    /// <summary>PDT-02</summary>
	{attribute 'OPC.UA.DA' := '1'}  				                
	sorbent_diff_pres_low												: REAL;
    /// <summary>PDT-02</summary>
	{attribute 'OPC.UA.DA' := '1'}  				                
	sorbent_diff_pres_high												: REAL;
    /// <summary>PDT-02</summary>
	{attribute 'OPC.UA.DA' := '1'}  				                
	sorbent_diff_pres_min												: REAL;
    /// <summary>PDT-02</summary>
	{attribute 'OPC.UA.DA' := '1'}  				                
	sorbent_diff_pres_offset											: REAL;

    /// <summary>PDT-03</summary>
	{attribute 'OPC.UA.DA' := '1'}  				                
	fan_diff_pres_low													: REAL;
    /// <summary>PDT-03</summary>
	{attribute 'OPC.UA.DA' := '1'}  				                
	fan_diff_pres_high													: REAL;
    /// <summary>PDT-03</summary>
	{attribute 'OPC.UA.DA' := '1'}  				                
	fan_diff_pres_min													: REAL;
    /// <summary>PDT-03</summary>
	{attribute 'OPC.UA.DA' := '1'}  				                
	fan_diff_pres_offset												: REAL;

    /// <summary>PT-01</summary>
	{attribute 'OPC.UA.DA' := '1'}  				                
	reactor_pres_low													: REAL;
    /// <summary>PT-01</summary>
	{attribute 'OPC.UA.DA' := '1'}  				                
	reactor_pres_high													: REAL;
    /// <summary>PT-01</summary>
	{attribute 'OPC.UA.DA' := '1'}  				                
	reactor_pres_min													: REAL;
    /// <summary>PT-01</summary>
	{attribute 'OPC.UA.DA' := '1'}  				                
	reactor_pres_offset													: REAL;

    /// <summary>TT-05</summary>
	{attribute 'OPC.UA.DA' := '1'}  				                
	reactor_wall_temp_offset											: REAL;

    /// <summary>TT-06</summary>
	{attribute 'OPC.UA.DA' := '1'}  				                
	outlet_line_temp_offset												: REAL;

	
    /// <summary>01-TT-01</summary>
	{attribute 'OPC.UA.DA' := '1'}  				                
	cart01_front_temp_offset											: REAL;
    /// <summary>10-TT-03</summary>
	{attribute 'OPC.UA.DA' := '1'}  				                
	cart01_back_temp_offset												: REAL;
    /// <summary>02-TT-01</summary>
	{attribute 'OPC.UA.DA' := '1'}  				                
	cart02_front_temp_offset											: REAL;
    /// <summary>02-TT-03</summary>
	{attribute 'OPC.UA.DA' := '1'}  				                
	cart02_back_temp_offset												: REAL;
    /// <summary>03-TT-01</summary>
	{attribute 'OPC.UA.DA' := '1'}  				                
	cart03_front_temp_offset											: REAL;
    /// <summary>03-TT-03</summary>
	{attribute 'OPC.UA.DA' := '1'}  				                
	cart03_back_temp_offset												: REAL;
    /// <summary>04-TT-01</summary>
	{attribute 'OPC.UA.DA' := '1'}  				                
	cart04_front_temp_offset											: REAL;
    /// <summary>04-TT-03</summary>
	{attribute 'OPC.UA.DA' := '1'}  				                
	cart04_back_temp_offset												: REAL;
    /// <summary>05-TT-01</summary>
	{attribute 'OPC.UA.DA' := '1'}  				                
	cart05_front_temp_offset											: REAL;
    /// <summary>05-TT-03</summary>
	{attribute 'OPC.UA.DA' := '1'}  				                
	cart05_back_temp_offset												: REAL;
    /// <summary>06-TT-01</summary>
	{attribute 'OPC.UA.DA' := '1'}  				                
	cart06_front_temp_offset											: REAL;
    /// <summary>06-TT-03</summary>
	{attribute 'OPC.UA.DA' := '1'}  				                
	cart06_back_temp_offset												: REAL;
    /// <summary>07-TT-01</summary>
	{attribute 'OPC.UA.DA' := '1'}  				                
	cart07_front_temp_offset											: REAL;
    /// <summary>07-TT-03</summary>
	{attribute 'OPC.UA.DA' := '1'}  				                
	cart07_back_temp_offset												: REAL;
    /// <summary>08-TT-01</summary>
	{attribute 'OPC.UA.DA' := '1'}  				                
	cart08_front_temp_offset											: REAL;
    /// <summary>08-TT-03</summary>
	{attribute 'OPC.UA.DA' := '1'}  				                
	cart08_back_temp_offset												: REAL;
    /// <summary>09-TT-01</summary>
	{attribute 'OPC.UA.DA' := '1'}  				                
	cart09_front_temp_offset											: REAL;
    /// <summary>09-TT-03</summary>
	{attribute 'OPC.UA.DA' := '1'}  				                
	cart09_back_temp_offset												: REAL;
    /// <summary>10-TT-01</summary>
	{attribute 'OPC.UA.DA' := '1'}  				                
	cart10_front_temp_offset											: REAL;
    /// <summary>10-TT-03</summary>
	{attribute 'OPC.UA.DA' := '1'}  				                
	cart10_back_temp_offset												: REAL;
    /// <summary>11-TT-01</summary>
	{attribute 'OPC.UA.DA' := '1'}  				                
	cart11_front_temp_offset											: REAL;
    /// <summary>11-TT-03</summary>
	{attribute 'OPC.UA.DA' := '1'}  				                
	cart11_back_temp_offset												: REAL;
    /// <summary>12-TT-01</summary>
	{attribute 'OPC.UA.DA' := '1'}  				                
	cart12_front_temp_offset											: REAL;
    /// <summary>12-TT-03</summary>
	{attribute 'OPC.UA.DA' := '1'}  				                
	cart12_back_temp_offset												: REAL;
	
END_VAR

// ---- GVLs/P0_Global_Variables.TcGVL
// Phase 0 - Global_Variables
// Rev 1.0 - May 11, 2024

VAR_GLOBAL

	sita_bits															: ARRAY[1..10] OF DINT;
	
	

	gbRS01TestError														: BOOL;
	gbRS02TestError														: BOOL;
	gbRS03TestError														: BOOL;
	
	gbDrainageOn														: BOOL;
	gbSafeShutdownRunning												: BOOL;

	giEvacuationErrorRS													: INT		:= 0;
	giDesorptionErrorRS													: INT		:= 0;
	giSafeShutdown1RS													: INT		:= 0;
	giSafeShutdown23RS													: INT		:= 0;
	
	gsCycleMode															: STRING;
	gsCycleStage														: STRING;
	gsM01RS01CycleStage													: STRING;
	gsM01RS02CycleStage													: STRING;
	gsM01RS03CycleStage													: STRING;
	
// These values allow points in error to be bypassed for testing purposes
	_BoilerOutletPresOff												: BOOL		:= TRUE;// FALSE;
	_BoilerOutletTempOff                        						: BOOL		:= FALSE;
	_CondensateCollectionTankFlowOff									: BOOL		:= FALSE;
	_CondensateCollectionTankLevelOff									: BOOL		:= FALSE;
	_CondensateCollectionTankO2Off										: BOOL		:= FALSE;
	_CondensateCollectionTankOutletLineTempOff  						: BOOL		:= FALSE;
	_CondensateCollectionTankPhOff										: BOOL		:= FALSE;
	_CondensateCollectionTankTempOff            						: BOOL		:= FALSE;
	_CondensateCollectionTankTurbidityOff								: BOOL		:= FALSE;
	_DeadAirFlowOff														: BOOL		:= FALSE;
	_DeadAirLineCo2Off													: BOOL		:= FALSE;
	_DeadAirLinePresOff													: BOOL		:= FALSE;
	_InstrumentAirCompPresOff                   						: BOOL		:= FALSE;
	_InstrumentAirCompTempOff                   						: BOOL		:= TRUE;
	_PostCondenserLinePresOff											: BOOL		:= FALSE;
	_PostCondenserLineTempOff                   						: BOOL		:= FALSE;
	_PreCondenserLinePresOff											: BOOL		:= FALSE;
	_PreCondenserLineTempOff                    						: BOOL		:= FALSE;
	_ProductCondensateDrumLevelOff										: BOOL		:= FALSE;
	_ProductCondenserPumpOutlerLiquidFlowOff							: BOOL		:= FALSE;
	_ProductCondenserPumpOutletTempOff          						: BOOL		:= FALSE;
	_ProductOutletCo2Off												: BOOL		:= FALSE;
	_ProductOutletH2oOff												: BOOL		:= FALSE;
	_ProductCo2SampleH2oOff												: BOOL		:= FALSE;
	_ProductOutletTemperatureOff										: BOOL		:= FALSE;
	_ProductOutletO2Off													: BOOL		:= FALSE;
	_ProductOutletPresOff												: BOOL		:= FALSE;
	_ProductOutletTempOff                       						: BOOL		:= FALSE;
	_ProductOutMassFlowOff												: BOOL		:= FALSE;
	_ProductOutVolumetricFlowOff										: BOOL		:= FALSE;
	_ProductVacuumPresOff												: BOOL		:= FALSE;
	_PurgeProductLinePresOff											: BOOL		:= FALSE;
	_PurgeProductLineTempOff											: BOOL		:= FALSE;
	_SteamHeadFlowOff													: BOOL		:= FALSE;
	_WaterToBoilerFlowOff												: BOOL		:= FALSE;
	_WeatherHumidityOff													: BOOL		:= FALSE;
	_WeatherNoiseLevelOff												: BOOL		:= FALSE;
	_WeatherPressureOff													: BOOL		:= FALSE;
	_WeatherTempOff														: BOOL		:= FALSE;
	_WeatherWindDirectionOff											: BOOL		:= FALSE;
	_WeatherWindSpeedOff												: BOOL		:= FALSE;

	_CondensateFlowOff													: BOOL		:= FALSE;
 	_SteamManifoldLinePresOff											: BOOL		:= FALSE;
	_SteamTempNearRS01Off												: BOOL		:= FALSE;           						
	_SteamTempNearRS03Off												: BOOL		:= FALSE;           						
	_CondensateTempOff													: BOOL		:= FALSE;           						
	
END_VAR

// ---- GVLs/m01.TcGVL
// Phase 0 - m01
// Rev 1.0 - April 25, 2024

{attribute 'qualified_only'}
VAR_GLOBAL

	{attribute 'OPC.UA.DA' := '1'}  				                
	{attribute 'OPC.UA.DA.Access' := '1'}  				                
	plc_version															: STRING;

	{attribute 'OPC.UA.DA' := '1'}  				                
	ts_Cycle_Mode														: STRING;		// Starts process based on each character in integer format
	{attribute 'OPC.UA.DA' := '1'}  				                
	tb_HMI_Active														: BOOL;			// An HMI program is running and communicating
	{attribute 'OPC.UA.DA' := '1'}  				                
	tb_Acknowledge_Alarm												: BOOL;			// Clears current alarm
	{attribute 'OPC.UA.DA' := '1'}  				                
	tb_Clear_Alarm_All													: BOOL;			// Clears current alarm
	{attribute 'OPC.UA.DA' := '1'}  				                
	tb_Cancel_Cycle														: BOOL;			// Complete current cycle then stop
	{attribute 'OPC.UA.DA' := '1'}  				                
	tb_Stop_Process														: BOOL;			// Stop current process immediately
	{attribute 'OPC.UA.DA' := '1'}  				                
	tb_Reset_Process													: BOOL;
	
	{attribute 'OPC.UA.DA' := '1'}  				                
	{attribute 'OPC.UA.DA.Access' := '1'}  				                
	tb_Alarm_Active														: BOOL;			// An alarm is active
	{attribute 'OPC.UA.DA' := '1'}  				                
	{attribute 'OPC.UA.DA.Access' := '1'}  				                
	ts_Alarm															: STRING;		// Active alarm string
	{attribute 'OPC.UA.DA' := '1'}  				                
	{attribute 'OPC.UA.DA.Access' := '1'}  				                
	ts_User_Message														: STRING;		// Message corresponding to active alarm
	{attribute 'OPC.UA.DA' := '1'}  				                
	{attribute 'OPC.UA.DA.Access' := '1'}  				                
	ti_Alarm_Severity													: INT;			// Alarm level (not implemented)	
	{attribute 'OPC.UA.DA' := '1'}  
	processAlarms														: ARRAY[0.._ALARM_COUNT] OF STRING;
	{attribute 'OPC.UA.DA' := '1'}  
	processAlarmsMessage												: ARRAY[0.._ALARM_COUNT] OF STRING;
					
	{attribute 'OPC.UA.DA' := '1'}  				                
	{attribute 'OPC.UA.DA.Access' := '1'}  				                
	tb_Auto_Mode_On														: BOOL;			// Machine is currently in auto mode
	
	
	
	{attribute 'OPC.UA.DA' := '1'} 	
	dispatch_active_queue_steam_pump 									: ARRAY[1..rs_count] OF UINT;
	{attribute 'OPC.UA.DA' := '1'} 	
	dispatch_passive_queue_steam_pump 									: ARRAY[1..rs_count] OF UINT;
		{attribute 'OPC.UA.DA' := '1'} 	
	dispatch_active_queue_dead_pump 									: ARRAY[1..rs_count] OF UINT; 
	{attribute 'OPC.UA.DA' := '1'} 	
	dispatch_passive_queue_dead_pump 									: ARRAY[1..rs_count] OF UINT; 

	
    /// <summary>FT-02</summary>
	{attribute 'OPC.UA.DA' := '1'}  				                
	{attribute 'OPC.UA.DA.Access' := '1'}  				                
	condensate_flow														: REAL;
    /// <summary>FT-02</summary>
	{attribute 'OPC.UA.DA' := '1'}  				                
	{attribute 'OPC.UA.DA.Access' := '1'}  				                
	condensate_flow_error										AT %I*	: BOOL;
    /// <summary>condensate flow</summary>
	FT_02														AT %I*	: INT;

    /// <summary>PT-02</summary>
	{attribute 'OPC.UA.DA' := '1'}  				                
	{attribute 'OPC.UA.DA.Access' := '1'}  				                
	steam_manifold_line_pres											: REAL;
    /// <summary>PT-02</summary>
	{attribute 'OPC.UA.DA' := '1'}  				                
	{attribute 'OPC.UA.DA.Access' := '1'}  				                
	steam_manifold_line_pres_error								AT %I*	: BOOL;
    /// <summary>steam manifold line pres</summary>
	PT_02														AT %I*	: INT;

    /// <summary>LS-03</summary>
	{attribute 'OPC.UA.DA' := '1'}  				                
	{attribute 'OPC.UA.DA.Access' := '1'}  				                
	condensate_from_cooling_and_purge_lines_lsl					AT %I*	: BOOL;
	
    /// <summary>LS-04</summary>
	{attribute 'OPC.UA.DA' := '1'}  				                
	{attribute 'OPC.UA.DA.Access' := '1'}  				                
	condensate_from_cooling_and_purge_lines_lsh					AT %I*	: BOOL;

    /// <summary>P-02</summary>
	{attribute 'OPC.UA.DA' := '1'}  				                
	condensate_from_cooling_and_purge_lines_pump						: BOOL;
    /// <summary>P-02</summary>
	{attribute 'OPC.UA.DA' := '1'}  				                
	{attribute 'OPC.UA.DA.Access' := '1'}  				                
	condensate_from_cooling_and_purge_lines_pump_cmd_status				: BOOL;
    /// <summary>condensate from cooling and purge lines pump</summary>
	P_02														AT %Q*	: BOOL;

    /// <summary>TT-10</summary>
	{attribute 'OPC.UA.DA' := '1'}  				                
	{attribute 'OPC.UA.DA.Access' := '1'}  				                
	steam_temp_near_rs1													: REAL;
    /// <summary>TT-10</summary>
	{attribute 'OPC.UA.DA' := '1'}  				                
	{attribute 'OPC.UA.DA.Access' := '1'}  				                
	steam_temp_near_rs1_error									AT %I*	: BOOL;
    /// <summary>steam temp near rs1 error</summary>
	TT_10														AT %I*	: INT;

    /// <summary>TT-11</summary>
	{attribute 'OPC.UA.DA' := '1'}  				                
	{attribute 'OPC.UA.DA.Access' := '1'}  				                
	steam_temp_near_rs3													: REAL;
    /// <summary>TT-11</summary>
	{attribute 'OPC.UA.DA' := '1'}  				                
	{attribute 'OPC.UA.DA.Access' := '1'}  				                
	steam_temp_near_rs3_error									AT %I*	: BOOL;
    /// <summary>steam temp near rs3 error</summary>
	TT_11														AT %I*	: INT;

    /// <summary>TT-12</summary>
	{attribute 'OPC.UA.DA' := '1'}  				                
	{attribute 'OPC.UA.DA.Access' := '1'}  				                
	condensate_temp														: REAL;
    /// <summary>TT-12</summary>
	{attribute 'OPC.UA.DA' := '1'}  				                
	{attribute 'OPC.UA.DA.Access' := '1'}  				                
	condensate_temp_error										AT %I*	: BOOL;
    /// <summary>condensate temp</summary>
	TT_12														AT %I*	: INT;

	{attribute 'OPC.UA.DA' := '1'}  				                
	l1_current															: REAL;
	{attribute 'OPC.UA.DA' := '1'}  				                
	l1_current_error											AT %I*	: BOOL;
	IT_01														AT %I*	: INT;
	{attribute 'OPC.UA.DA' := '1'}  				                
	l2_current															: REAL;
	{attribute 'OPC.UA.DA' := '1'}  				                
	l2_current_error											AT %I*	: BOOL;
	IT_02														AT %I*	: INT;
	{attribute 'OPC.UA.DA' := '1'}  				                
	l3_current															: REAL;
	{attribute 'OPC.UA.DA' := '1'}  				                
	l3_current_error											AT %I*	: BOOL;
	IT_03														AT %I*	: INT;
	
	{attribute 'OPC.UA.DA' := '1'}  				                
	l1_voltage															: REAL;
	{attribute 'OPC.UA.DA' := '1'}  				                
	l1_volatge_error											AT %I*	: BOOL;
	VT_01														AT %I*	: INT;
	{attribute 'OPC.UA.DA' := '1'}  				                
	l2_voltage															: REAL;
	{attribute 'OPC.UA.DA' := '1'}  				                
	l2_volatge_error											AT %I*	: BOOL;
	VT_02														AT %I*	: INT;
	{attribute 'OPC.UA.DA' := '1'}  				                
	l3_voltage															: REAL;
	{attribute 'OPC.UA.DA' := '1'}  				                
	l3_volatge_error											AT %I*	: BOOL;
	VT_03														AT %I*	: INT;

END_VAR

VAR_GLOBAL PERSISTENT

	/// SCALING
	
    /// <summary>FT-02</summary>
	{attribute 'OPC.UA.DA' := '1'}  				                
	condensate_flow_low													: REAL;
    /// <summary>FT-02</summary>
	{attribute 'OPC.UA.DA' := '1'}  				                
	condensate_flow_high												: REAL;
    /// <summary>FT-02</summary>
	{attribute 'OPC.UA.DA' := '1'}  				                
	condensate_flow_min													: REAL;
    /// <summary>FT-02</summary>
	{attribute 'OPC.UA.DA' := '1'}  				                
	condensate_flow_offset												: REAL;

    /// <summary>PT-02</summary>
	{attribute 'OPC.UA.DA' := '1'}  				                
	steam_manifold_line_pres_low										: REAL;
    /// <summary>PT-02</summary>
	{attribute 'OPC.UA.DA' := '1'}  				                
	steam_manifold_line_pres_high										: REAL;
    /// <summary>PT-02</summary>
	{attribute 'OPC.UA.DA' := '1'}  				                
	steam_manifold_line_pres_min										: REAL;
    /// <summary>PT-02</summary>
	{attribute 'OPC.UA.DA' := '1'}  				                
	steam_manifold_line_pres_offset										: REAL;

    /// <summary>TT-10</summary>
	{attribute 'OPC.UA.DA' := '1'}  				                
	steam_temp_near_rs1_offset											: REAL;

    /// <summary>TT-11</summary>
	{attribute 'OPC.UA.DA' := '1'}  				                
	steam_temp_near_rs3_offset											: REAL;
	
    /// <summary>TT-12</summary>
	{attribute 'OPC.UA.DA' := '1'}  				                
	condensate_temp_offset												: REAL;

	
	/// SET POINTS

	{attribute 'OPC.UA.DA' := '1'}
	SP_adsorption_sorbent_hightemp_startco2analyzer						: REAL;		

	{attribute 'OPC.UA.DA' := '1'}
	SP_adsorption_outletco2_highlimit									: REAL;		

	{attribute 'OPC.UA.DA' := '1'}
	SP_repres_preslimit_clampsretract									: REAL;		

	{attribute 'OPC.UA.DA' := '1'}
	SP_clampsretract_timedelay											: REAL;		

	{attribute 'OPC.UA.DA' := '1'}
	SP_repres_pres_highlimit											: REAL;		

	{attribute 'OPC.UA.DA' := '1'}
	SP_doorsopenclose_timedelay											: REAL;		


	
	{attribute 'OPC.UA.DA' := '1'}
	SP_adsorption_duration												: REAL;
	{attribute 'OPC.UA.DA' := '1'}
	SP_adsorption_valve_max_retries										: INT;		
	{attribute 'OPC.UA.DA' := '1'}
	SP_adsorption_valve_rotational_velocity								: REAL;		
	{attribute 'OPC.UA.DA' := '1'}
	SP_ambient_pressure													: REAL;
	{attribute 'OPC.UA.DA' := '1'}
	SP_cycle_start_offset_duration										: REAL;
	{attribute 'OPC.UA.DA' := '1'}
	SP_dead_time_in_cycle_duration										: REAL;
	{attribute 'OPC.UA.DA' := '1'}
	SP_desired_cycle_count												: INT;
	{attribute 'OPC.UA.DA' := '1'}
	SP_evacuation_duration												: REAL;
	{attribute 'OPC.UA.DA' := '1'}
	SP_evacuation_ideal_pressure										: REAL;
	{attribute 'OPC.UA.DA' := '1'}
	SP_evacuation_unacceptable_pressure									: REAL;
	{attribute 'OPC.UA.DA' := '1'}
	SP_include_reactor_set_1_in_process									: BOOL;					
	{attribute 'OPC.UA.DA' := '1'}
	SP_include_reactor_set_2_in_process									: BOOL;
	{attribute 'OPC.UA.DA' := '1'}
	SP_include_reactor_set_3_in_process									: BOOL;	
	{attribute 'OPC.UA.DA' := '1'}
	SP_initial_maximum_steam_valve_percent_open							: REAL;
	{attribute 'OPC.UA.DA' := '1'}
	SP_initial_steam_purge_reactor_pressure								: REAL;
	{attribute 'OPC.UA.DA' := '1'}
	SP_leak_test_duration												: REAL;
	{attribute 'OPC.UA.DA' := '1'}
	SP_maximum_desorption_starting_pressure								: REAL;							
	{attribute 'OPC.UA.DA' := '1'}
	SP_maximum_inlet_air_temperature_during_adsorption					: REAL;						
	{attribute 'OPC.UA.DA' := '1'}
	SP_maximum_safe_reactor_steam_pressure								: REAL;
	{attribute 'OPC.UA.DA' := '1'}
	SP_maximum_sorbent_temperature_during_desorption					: REAL;			
	{attribute 'OPC.UA.DA' := '1'}
	SP_maximum_target_sorbent_temperature_during_purge					: REAL;												// PS 04_25_24			
	{attribute 'OPC.UA.DA' := '1'}
	SP_maximum_target_steam_pressure									: REAL;			
	{attribute 'OPC.UA.DA' := '1'}
	SP_minimum_desired_inlet_co2_concentration_during_adsorption		: REAL;						
	{attribute 'OPC.UA.DA' := '1'}
	SP_minimum_inlet_air_temperature_during_adsorption					: REAL;						
	{attribute 'OPC.UA.DA' := '1'}
	SP_module_steam_line_high_pressure									: REAL;
	{attribute 'OPC.UA.DA' := '1'}
	SP_module_steam_line_high_temperature								: REAL;
	{attribute 'OPC.UA.DA' := '1'}
	SP_module_steam_line_low_pressure									: REAL;
	{attribute 'OPC.UA.DA' := '1'}
	SP_module_steam_line_low_temperature								: REAL;
	{attribute 'OPC.UA.DA' := '1'}
	SP_percent_from_steam_purge_target_pressure							: REAL;
	{attribute 'OPC.UA.DA' := '1'}
	SP_percent_of_ambient_pressure										: REAL;
	{attribute 'OPC.UA.DA' := '1'}
	SP_reactor_set_1_vfd_percent										: INT;
	{attribute 'OPC.UA.DA' := '1'}
	SP_reactor_set_2_vfd_percent										: INT;
	{attribute 'OPC.UA.DA' := '1'}
	SP_reactor_set_3_vfd_percent										: INT;
	{attribute 'OPC.UA.DA' := '1'}
	SP_repressurization_duration										: REAL;
	{attribute 'OPC.UA.DA' := '1'}
	SP_start_steam_purge_reactor_pressure								: REAL;
	{attribute 'OPC.UA.DA' := '1'}
	SP_steam_pressure_control_valve_initial_opening_duration			: REAL;					
	{attribute 'OPC.UA.DA' := '1'}
	SP_steam_pressurization_and_purge_duration							: REAL;						
	{attribute 'OPC.UA.DA' := '1'}
	SP_steam_purge_pressure												: REAL;
	{attribute 'OPC.UA.DA' := '1'}
	SP_steam_purge_pressure_decrease									: REAL;												// PS 04_25_24
	{attribute 'OPC.UA.DA' := '1'}
	SP_target_desorption_starting_pressure								: REAL;
	{attribute 'OPC.UA.DA' := '1'}
	SP_target_duration_from_adsorption_start_until_sorbent_cool			: REAL;							
	{attribute 'OPC.UA.DA' := '1'}
	SP_target_pressure_change											: REAL;
	{attribute 'OPC.UA.DA' := '1'}
	SP_unacceptable_duration_from_adsorption_start_until_sorbent_cool	: REAL;					
	{attribute 'OPC.UA.DA' := '1'}
	SP_unacceptable_pressure_change										: REAL;
	{attribute 'OPC.UA.DA' := '1'}
	SP_undesirable_duration_from_adsorption_start_until_sorbent_cool	: REAL;
	{attribute 'OPC.UA.DA' := '1'}
	SP_vacuum_assisted_purge											: BOOL;
	{attribute 'OPC.UA.DA' := '1'}
	SP_vacuum_cooling_duration											: REAL;
	{attribute 'OPC.UA.DA' := '1'}
	SP_vacuum_cooling_target_pressure									: REAL;
	{attribute 'OPC.UA.DA' := '1'}
	SP_vacuum_cooling_target_temperature								: REAL;
	{attribute 'OPC.UA.DA' := '1'}
	SP_vacuum_cooling_unacceptable_pressure								: REAL;
	{attribute 'OPC.UA.DA' := '1'}
	SP_vacuum_cooling_unacceptable_temperature							: REAL;
	{attribute 'OPC.UA.DA' := '1'}
	SP_extend_wallace_clamp_duration									: REAL;
			
END_VAR

// ---- GVLs/m01_rs1.TcGVL
// Phase 0 - m01_rs1
// Rev 1.0 - April 24, 2024

{attribute 'qualified_only'}
VAR_GLOBAL
 
	{attribute 'OPC.UA.DA' := '1'}  				                
	{attribute 'OPC.UA.DA.Access' := '1'}  				                
	ti_Total_Cycle_Count												: DINT; 
	{attribute 'OPC.UA.DA' := '1'}  				                
	{attribute 'OPC.UA.DA.Access' := '1'}  				                
	ti_Cycle_Count														: INT; 
	{attribute 'OPC.UA.DA' := '1'}  				                
	{attribute 'OPC.UA.DA.Access' := '1'}  				                
	ti_Machine_State													: INT;
	{attribute 'OPC.UA.DA' := '1'}  				                
	{attribute 'OPC.UA.DA.Access' := '1'}  				                
	ti_Current_Step														: INT;
	{attribute 'OPC.UA.DA' := '1'}  				                
	{attribute 'OPC.UA.DA.Access' := '1'}  				                
	tb_Process_Running													: BOOL;
	{attribute 'OPC.UA.DA' := '1'}  				                
	{attribute 'OPC.UA.DA.Access' := '1'}  				                
	tb_Repressurization_Running											: BOOL;
	{attribute 'OPC.UA.DA' := '1'}  				                
	{attribute 'OPC.UA.DA.Access' := '1'}  				                
	tb_Adsorption_Running												: BOOL;
	{attribute 'OPC.UA.DA' := '1'}  				                
	{attribute 'OPC.UA.DA.Access' := '1'}  				                
	tb_Evacuation_Running												: BOOL;
	{attribute 'OPC.UA.DA' := '1'}  				                
	{attribute 'OPC.UA.DA.Access' := '1'}  				                
	tb_Desorption_Running												: BOOL;
	{attribute 'OPC.UA.DA' := '1'}  				                
	{attribute 'OPC.UA.DA.Access' := '1'}  				                
	tb_Process_Complete													: BOOL;
	{attribute 'OPC.UA.DA' := '1'}  				                
	{attribute 'OPC.UA.DA.Access' := '1'}  				                
	tr_Remaining_Time													: REAL;
	{attribute 'OPC.UA.DA' := '1'}  				                
	{attribute 'OPC.UA.DA.Access' := '1'}  				                
	ti_Status															: INT;
	{attribute 'OPC.UA.DA' := '1'}  				                
	{attribute 'OPC.UA.DA.Access' := '1'}  				                
	ts_Status_Text														: STRING;		

	
	{attribute 'OPC.UA.DA' := '1'}  				                
	{attribute 'OPC.UA.DA.Access' := '1'}  				                
	cycle_stage															: STRING;


    /// <summary>PWR-01</summary>
	{attribute 'OPC.UA.DA' := '1'}  				                
	power_control														: BOOL;
    /// <summary>PWR-01</summary>
	{attribute 'OPC.UA.DA' := '1'}  				                
	{attribute 'OPC.UA.DA.Access' := '1'}  				                
	power_control_status												: BOOL;
    /// <summary>power_cmd</summary>
	PWR_01														AT %Q*	: BOOL;
	circuit_breaker_no_feedback									AT %I*	: BOOL;
	circuit_breaker_nc_feedback									AT %I*	: BOOL;
	
    /// <summary>LS-01</summary>
	{attribute 'OPC.UA.DA' := '1'}  				                
	{attribute 'OPC.UA.DA.Access' := '1'}  				                
	condensate_lsl												AT %I*	: BOOL;
	
    /// <summary>LS-02</summary>
	{attribute 'OPC.UA.DA' := '1'}  				                
	{attribute 'OPC.UA.DA.Access' := '1'}  				                
	condensate_lsh												AT %I*	: BOOL;

    /// <summary>P-01</summary>
	{attribute 'OPC.UA.DA' := '1'}  				                
	condensate_pump														: BOOL;
    /// <summary>P-01</summary>
	{attribute 'OPC.UA.DA' := '1'}  				                
	{attribute 'OPC.UA.DA.Access' := '1'}  				                
	condensate_pump_cmd_status											: BOOL;
    /// <summary>condensate pump</summary>
	P_01														AT %Q*	: BOOL;

    /// <summary>RS_PCV-01</summary>
	{attribute 'OPC.UA.DA' := '1'}  				                
	steam_control_valve													: REAL;
    /// <summary>RS_PCV-01</summary>
	{attribute 'OPC.UA.DA' := '1'}  				                
	{attribute 'OPC.UA.DA.Access' := '1'}  				                
	steam_control_valve_position										: REAL;
    /// <summary>rs steam control valve</summary>
	PCV_01														AT %Q*	: INT;
    /// <summary>rs steam control valve</summary>
	PCV_01_position												AT %I*	: INT;
    /// <summary>RS_PCV-01</summary>
	{attribute 'OPC.UA.DA' := '1'}  				                
	{attribute 'OPC.UA.DA.Access' := '1'}  				                
	steam_control_valve_position_error							AT %I*	: BOOL;
    /// <summary>RS_PCV-01</summary>                  	           
	{attribute 'OPC.UA.DA' := '1'}  				                
	steam_control_valve_mode											: INT;			
    /// <summary>PCV-01</summary>                  	           
	{attribute 'OPC.UA.DA' := '1'}  				                
	{attribute 'OPC.UA.DA.Access' := '1'}  				                
	steam_control_valve_current_mode									: INT;			
    /// <summary>PCV-01</summary>                  	           
	steam_control_valve_kp												: REAL		:= 0.01; 
    /// <summary>PCV-01</summary>                  	           
	steam_control_valve_ki												: REAL		:= 0.01;
    /// <summary>PCV-01</summary>                  	           
	steam_control_valve_loop_time										: REAL		:= 2000;
    /// <summary>PCV-01</summary>                  	           
	steam_control_valve_iband											: REAL		:= 6;
    /// <summary>PCV-01</summary>                  	           
	steam_control_valve_base											: INT		:= 13110;
    /// <summary>PCV-01</summary>                  	           
	steam_control_valve_base_adjust										: INT		:= 10;
		                                	        	
    /// <summary>XV-04</summary>
	{attribute 'OPC.UA.DA' := '1'}  				                
	dead_air_valve														: BOOL;
    /// <summary>XV-04</summary>
	{attribute 'OPC.UA.DA' := '1'}  				                
	{attribute 'OPC.UA.DA.Access' := '1'}  				                
	dead_air_valve_open_cmd_status										: BOOL;
    /// <summary>XV-04</summary>
	{attribute 'OPC.UA.DA' := '1'}  				                
	{attribute 'OPC.UA.DA.Access' := '1'}  				                
	dead_air_valve_open											AT %I*	: BOOL;
    /// <summary>XV-04</summary>
	{attribute 'OPC.UA.DA' := '1'}  				                
	{attribute 'OPC.UA.DA.Access' := '1'}  				                
	dead_air_valve_closed										AT %I*	: BOOL;
    /// <summary>dead air valve</summary>
	XV_04														AT %Q*	: BOOL;
	
    /// <summary>RS_XV-05</summary>
	{attribute 'OPC.UA.DA' := '1'}  				                
	purge_valve															: BOOL;
    /// <summary>RS_XV-05</summary>
	{attribute 'OPC.UA.DA' := '1'}  				                
	{attribute 'OPC.UA.DA.Access' := '1'}  				                
	purge_valve_open_cmd_status											: BOOL;
    /// <summary>RS_XV-05</summary>
	{attribute 'OPC.UA.DA' := '1'}  				                
	{attribute 'OPC.UA.DA.Access' := '1'}  				                
	purge_valve_open											AT %I*	: BOOL;
    /// <summary>RS_XV-05</summary>
	{attribute 'OPC.UA.DA' := '1'}  				                
	{attribute 'OPC.UA.DA.Access' := '1'}  				                
	purge_valve_closed											AT %I*	: BOOL;
    /// <summary>rs purge valve</summary>
	XV_05														AT %Q*	: BOOL;
	
    /// <summary>XV-06</summary>
	{attribute 'OPC.UA.DA' := '1'}  				                
	cooling_valve														: BOOL;
    /// <summary>XV-06</summary>
	{attribute 'OPC.UA.DA' := '1'}  				                
	{attribute 'OPC.UA.DA.Access' := '1'}  				                
	cooling_valve_open_cmd_status										: BOOL;
    /// <summary>XV-06</summary>
	{attribute 'OPC.UA.DA' := '1'}  				                
	{attribute 'OPC.UA.DA.Access' := '1'}  				                
	cooling_valve_open											AT %I*	: BOOL;
    /// <summary>XV-06</summary>
	{attribute 'OPC.UA.DA' := '1'}  				                
	{attribute 'OPC.UA.DA.Access' := '1'}  				                
	cooling_valve_closed										AT %I*	: BOOL;
    /// <summary>cooling valve</summary>
	XV_06														AT %Q*	: BOOL;
	
    /// <summary>XV-07</summary>
	{attribute 'OPC.UA.DA' := '1'}  				                
	steam_header_valve													: BOOL;
    /// <summary>XV-07</summary>
	{attribute 'OPC.UA.DA' := '1'}  				                
	{attribute 'OPC.UA.DA.Access' := '1'}  				                
	steam_header_valve_open_cmd_status									: BOOL;
    /// <summary>XV-07</summary>
	{attribute 'OPC.UA.DA' := '1'}  				                
	{attribute 'OPC.UA.DA.Access' := '1'}  				                
	steam_header_valve_open										AT %I*	: BOOL;
    /// <summary>XV-07</summary>
	{attribute 'OPC.UA.DA' := '1'}  				                
	{attribute 'OPC.UA.DA.Access' := '1'}  				                
	steam_header_valve_closed									AT %I*	: BOOL;
    /// <summary>steam header valve</summary>
	XV_07														AT %Q*	: BOOL;

END_VAR

// ---- GVLs/m01_rs1_r1.TcGVL
// Phase 0 - m01_rs1_r1
// Rev 1.0 - April 11, 2024

{attribute 'qualified_only'}
VAR_GLOBAL

    /// <summary>AT-01</summary>																		// Summary defines hover over text while in twincat 3 program
	{attribute 'OPC.UA.DA' := '1'}  				                									// OPC_UA tag
	{attribute 'OPC.UA.DA.Access' := '1'}																// OPC_UA tag definition - '1' indicates Read Only, '2' indicates Write Only (not used), '3' indicates Read Write (default)  				                
	inlet_co2															: REAL;							// Tag value to read (scaled)
    /// <summary>AT-01</summary>
	{attribute 'OPC.UA.DA' := '1'}  				                
	{attribute 'OPC.UA.DA.Access' := '1'}  				                
	inlet_co2_error												AT %I*	: BOOL;							// Combination OPC_UA tag and twincat input variable
    /// <summary>Inlet CO2</summary>
	AT_01														AT %I*	: INT;							// Raw input data from sensor - not available as tag

    /// <summary>AT-01_pump</summary>
	{attribute 'OPC.UA.DA' := '1'}  				                
	inlet_co2_pump														: BOOL;
    /// <summary>AT-01_pump</summary>
	{attribute 'OPC.UA.DA' := '1'}  				                
	{attribute 'OPC.UA.DA.Access' := '1'}  				                
	inlet_co2_pump_cmd_status											: BOOL;
    /// <summary>Inlet CO2 pump</summary>
	AT_01_pump													AT %Q*	: BOOL;
    /// <summary>AT-01_solenoid</summary>
	{attribute 'OPC.UA.DA' := '1'}  				                
	inlet_co2_sol														: BOOL;
    /// <summary>AT-01_solenoid</summary>
	{attribute 'OPC.UA.DA' := '1'}  				                
	{attribute 'OPC.UA.DA.Access' := '1'}  				                
	inlet_co2_sol_cmd_status											: BOOL;
    /// <summary>Inlet CO2 solenoid</summary>
	AT_01_sol													AT %Q*	: BOOL;

    /// <summary>AT-02</summary>
	{attribute 'OPC.UA.DA' := '1'}  				                
	{attribute 'OPC.UA.DA.Access' := '1'}  				                
	inlet_h2o															: REAL;
    /// <summary>AT-02</summary>
	{attribute 'OPC.UA.DA' := '1'}  				                
	{attribute 'OPC.UA.DA.Access' := '1'}  				                
	inlet_h2o_error												AT %I*	: BOOL;
    /// <summary>Inlet H20</summary>
	AT_02														AT %I*	: INT;

    /// <summary>AT-03</summary>
	{attribute 'OPC.UA.DA' := '1'}  				                
	{attribute 'OPC.UA.DA.Access' := '1'}  				                
	outlet_co2															: REAL;
    /// <summary>AT-03</summary>
	{attribute 'OPC.UA.DA' := '1'}  				                
	{attribute 'OPC.UA.DA.Access' := '1'}  				                
	outlet_co2_error											AT %I*	: BOOL;
    /// <summary>Outlet CO2</summary>
	AT_03														AT %I*	: INT;
	
    /// <summary>AT-03_pump</summary>
	{attribute 'OPC.UA.DA' := '1'}  				                
	outlet_co2_pump														: BOOL;
    /// <summary>AT-03_pump</summary>
	{attribute 'OPC.UA.DA' := '1'}  				                
	{attribute 'OPC.UA.DA.Access' := '1'}  				                
	outlet_co2_pump_cmd_status											: BOOL;
    /// <summary>Inlet CO2 pump</summary>
	AT_03_pump													AT %Q*	: BOOL;
    /// <summary>AT-03_solenoid</summary>
	{attribute 'OPC.UA.DA' := '1'}  				                
	outlet_co2_sol														: BOOL;
    /// <summary>AT-03_solenoid</summary>
	{attribute 'OPC.UA.DA' := '1'}  				                
	{attribute 'OPC.UA.DA.Access' := '1'}  				                
	outlet_co2_sol_cmd_status											: BOOL;
    /// <summary>Outlet CO2 solenoid</summary>
	AT_03_sol													AT %Q*	: BOOL;

    /// <summary>AT-04</summary>
	{attribute 'OPC.UA.DA' := '1'}  				                
	{attribute 'OPC.UA.DA.Access' := '1'}  				                
	outlet_h2o															: REAL;
    /// <summary>AT-04</summary>
	{attribute 'OPC.UA.DA' := '1'}  				                
	{attribute 'OPC.UA.DA.Access' := '1'}  				                
	outlet_h2o_error											AT %I*	: BOOL;
    /// <summary>Outlet H20</summary>
	AT_04														AT %I*	: INT;

    /// <summary>FT-01</summary>
	{attribute 'OPC.UA.DA' := '1'}  				                
	{attribute 'OPC.UA.DA.Access' := '1'}  				                
	air_flow															: REAL;
    /// <summary>FT-01</summary>
	{attribute 'OPC.UA.DA' := '1'}  				                
	{attribute 'OPC.UA.DA.Access' := '1'}  				                
	air_flow_error												AT %I*	: BOOL;
    /// <summary>Air flow</summary>
	FT_01														AT %I*	: INT;
	
    /// <summary>PDT-01</summary>
	{attribute 'OPC.UA.DA' := '1'}  				                
	{attribute 'OPC.UA.DA.Access' := '1'}  				                
	filter_diff_pres													: REAL;
    /// <summary>PDT-01</summary>
	{attribute 'OPC.UA.DA' := '1'}  				                
	{attribute 'OPC.UA.DA.Access' := '1'}  				                
	filter_diff_pres_error										AT %I*	: BOOL;
    /// <summary>Filter diff pres</summary>
	PDT_01														AT %I*	: INT;

    /// <summary>PDT-02</summary>
	{attribute 'OPC.UA.DA' := '1'}  				                
	{attribute 'OPC.UA.DA.Access' := '1'}  				                
	sorbent_diff_pres													: REAL;
    /// <summary>PDT-02</summary>
	{attribute 'OPC.UA.DA' := '1'}  				                
	{attribute 'OPC.UA.DA.Access' := '1'}  				                
	sorbent_diff_pres_error										AT %I*	: BOOL;
    /// <summary>Sorbent diff pres</summary>
	PDT_02														AT %I*	: INT;

    /// <summary>PDT-03</summary>
	{attribute 'OPC.UA.DA' := '1'}  				                
	{attribute 'OPC.UA.DA.Access' := '1'}  				                
	fan_diff_pres														: REAL;
    /// <summary>PDT-03</summary>
	{attribute 'OPC.UA.DA' := '1'}  				                
	{attribute 'OPC.UA.DA.Access' := '1'}  				                
	fan_diff_pres_error											AT %I*	: BOOL;
    /// <summary>fan diff pres</summary>
	PDT_03														AT %I*	: INT;

     /// <summary>PT-01</summary>
	{attribute 'OPC.UA.DA' := '1'}  				                
	{attribute 'OPC.UA.DA.Access' := '1'}  				                
	reactor_pres														: REAL;
    /// <summary>PT-01</summary>
	{attribute 'OPC.UA.DA' := '1'}  				                
	{attribute 'OPC.UA.DA.Access' := '1'}  				                
	reactor_pres_error											AT %I*	: BOOL;
    /// <summary>Reactor pressure</summary>
	PT_01														AT %I*	: INT;

    /// <summary>TT-05</summary>
	{attribute 'OPC.UA.DA' := '1'}  				                
	{attribute 'OPC.UA.DA.Access' := '1'}  				                
	reactor_wall_temp													: REAL;
    /// <summary>Reactor wall temp</summary>
	{attribute 'OPC.UA.DA' := '1'}  				                
	{attribute 'OPC.UA.DA.Access' := '1'}  				                
	reactor_wall_temp_error										AT %I*	: BOOL;
    /// <summary>Reactor wall temp</summary>
	TT_05														AT %I*	: INT;
	
    /// <summary>TT-06</summary>
	{attribute 'OPC.UA.DA' := '1'}  				                
	{attribute 'OPC.UA.DA.Access' := '1'}  				                
	outlet_line_temp													: REAL;
    /// <summary>Outlet line temp</summary>
	{attribute 'OPC.UA.DA' := '1'}  				                
	{attribute 'OPC.UA.DA.Access' := '1'}  				                
	outlet_line_temp_error										AT %I*	: BOOL;
    /// <summary>Outlet_line temp</summary>
	TT_06														AT %I*	: INT;
	
	{attribute 'OPC.UA.DA' := '1'}  				                
	fan_vfd_enable														: BOOL :=  TRUE;
	{attribute 'OPC.UA.DA' := '1'}  				                
	fan_vfd_reset														: BOOL;
	{attribute 'OPC.UA.DA' := '1'}  				                
	{attribute 'OPC.UA.DA.Access' := '1'}  				                
	fan_vfd_enabled														: BOOL;
	{attribute 'OPC.UA.DA' := '1'}  				                
	{attribute 'OPC.UA.DA.Access' := '1'}  				                
	fan_vfd_error														: BOOL;
	{attribute 'OPC.UA.DA' := '1'}  				                
	fan_vfd																: REAL;
	{attribute 'OPC.UA.DA' := '1'}  				                
	{attribute 'OPC.UA.DA.Access' := '1'}  				                
	fan_vfd_input														: REAL;
	{attribute 'OPC.UA.DA' := '1'}  				                
	{attribute 'OPC.UA.DA.Access' := '1'}  				                
	fan_vfd_output														: REAL;
	{attribute 'OPC.UA.DA' := '1'}  				                
	{attribute 'OPC.UA.DA.Access' := '1'}  				                
	fan_vfd_output_current												: REAL;
	{attribute 'OPC.UA.DA' := '1'}  				                
	{attribute 'OPC.UA.DA.Access' := '1'}  				                
	fan_vfd_temperature													: REAL;
	fan_vfd_control												AT %Q*	: WORD;
	fan_vfd_target_vel											AT %Q*	: WORD;
	fan_vfd_status												AT %I*	: WORD;
	fan_vfd_velocity											AT %I*	: WORD;
	fan_vfd_ecat_state											AT %I*  : BOOL;
	fan_vfd_current												AT %I*	: DINT;
	fan_vfd_temp												AT %I*	: INT;

    /// <summary>XV-01 Both</summary>
	{attribute 'OPC.UA.DA' := '1'}  				                
	inlet_door_open														: BOOL;
    /// <summary>XV-01 Both</summary>
	{attribute 'OPC.UA.DA' := '1'}  				                
	inlet_door_close													: BOOL;
    /// <summary>XV-01 Left</summary>
	{attribute 'OPC.UA.DA' := '1'}  				                
	{attribute 'OPC.UA.DA.Access' := '1'}  				                
	inlet_door_left_open_ls										AT %I*	: BOOL;
    /// <summary>XV-01 Left</summary>
	{attribute 'OPC.UA.DA' := '1'}  				                
	{attribute 'OPC.UA.DA.Access' := '1'}  				                
	inlet_door_left_closed_ls									AT %I*	: BOOL;
    /// <summary>XV-01 Right</summary>
	{attribute 'OPC.UA.DA' := '1'}  				                
	{attribute 'OPC.UA.DA.Access' := '1'}  				                
	inlet_door_right_open_ls									AT %I*	: BOOL;
    /// <summary>XV-01 Right</summary>
	{attribute 'OPC.UA.DA' := '1'}  				                
	{attribute 'OPC.UA.DA.Access' := '1'}  				                
	inlet_door_right_closed_ls									AT %I*	: BOOL;
    /// <summary>Inlet Door</summary>
	XV_01_Door_Open_Solenoid_Valve								AT %Q*	: BOOL;
    /// <summary>Inlet Door</summary>
	XV_01_Door_Close_Solenoid_Valve								AT %Q*	: BOOL;
	
    /// <summary>XV-03 Both</summary>
	{attribute 'OPC.UA.DA' := '1'}  				                
	outlet_door_open													: BOOL;
    /// <summary>XV-03 Both</summary>
	{attribute 'OPC.UA.DA' := '1'}  				                
	outlet_door_close													: BOOL;
    /// <summary>XV-03 Left</summary>
	{attribute 'OPC.UA.DA' := '1'}  				                
	{attribute 'OPC.UA.DA.Access' := '1'}  				                
	outlet_door_left_open_ls									AT %I*	: BOOL;
    /// <summary>XV-03 Left</summary>
	{attribute 'OPC.UA.DA' := '1'}  				                
	{attribute 'OPC.UA.DA.Access' := '1'}  				                
	outlet_door_left_closed_ls									AT %I*	: BOOL;
    /// <summary>XV-03 Right</summary>
	{attribute 'OPC.UA.DA' := '1'}  				                
	{attribute 'OPC.UA.DA.Access' := '1'}  				                
	outlet_door_right_open_ls									AT %I*	: BOOL;
    /// <summary>XV-03 Right</summary>
	{attribute 'OPC.UA.DA' := '1'}  				                
	{attribute 'OPC.UA.DA.Access' := '1'}  				                
	outlet_door_right_closed_ls									AT %I*	: BOOL;
    /// <summary>Outlet Door</summary>
	XV_03_Door_Open_Solenoid_Valve								AT %Q*	: BOOL;
    /// <summary>Outlet Door</summary>
	XV_03_Door_Close_Solenoid_Valve								AT %Q*	: BOOL;

    /// <summary>XV-01 Both</summary>
	{attribute 'OPC.UA.DA' := '1'}  				                
	inlet_door_clamps_extend											: BOOL;
    /// <summary>XV-01 Both</summary>
	{attribute 'OPC.UA.DA' := '1'}  				                
	inlet_door_clamps_retract											: BOOL;
    /// <summary>XV-01 Left</summary>
	{attribute 'OPC.UA.DA' := '1'}  				                
	{attribute 'OPC.UA.DA.Access' := '1'}  				                
	inlet_door_left_clamps_extended_ls							AT %I*	: BOOL;
    /// <summary>XV-01 Right</summary>
	{attribute 'OPC.UA.DA' := '1'}  				                
	{attribute 'OPC.UA.DA.Access' := '1'}  				                
	inlet_door_right_clamps_extended_ls							AT %I*	: BOOL;
    /// <summary>Inlet Clamps</summary>
	XV_01_Left_Retract_Solenoid_Valve							AT %Q*	: BOOL;
    /// <summary>Inlet Clamps</summary>
	XV_01_Left_Extend_Solenoid_Valve							AT %Q*	: BOOL;
    /// <summary>Inlet Clamps</summary>
	XV_01_Right_Retract_Solenoid_Valve							AT %Q*	: BOOL;
    /// <summary>Inlet Clamps</summary>
	XV_01_Right_Extend_Solenoid_Valve							AT %Q*	: BOOL;

    /// <summary>XV-03 Both</summary>
	{attribute 'OPC.UA.DA' := '1'}  				                
	outlet_door_clamps_extend											: BOOL;
    /// <summary>XV-03 Both</summary>
	{attribute 'OPC.UA.DA' := '1'}  				                
	outlet_door_clamps_retract											: BOOL;
    /// <summary>XV-03 Left</summary>
	{attribute 'OPC.UA.DA' := '1'}  				                
	{attribute 'OPC.UA.DA.Access' := '1'}  				                
	outlet_door_left_clamps_extended_ls							AT %I*	: BOOL;
    /// <summary>XV-03 Right</summary>
	{attribute 'OPC.UA.DA' := '1'}  				                
	{attribute 'OPC.UA.DA.Access' := '1'}  				                
	outlet_door_right_clamps_extended_ls						AT %I*	: BOOL;
    /// <summary>Outlet Clamps</summary>
	XV_03_Left_Retract_Solenoid_Valve							AT %Q*	: BOOL;
    /// <summary>Outlet Clamps</summary>
	XV_03_Left_Extend_Solenoid_Valve							AT %Q*	: BOOL;
    /// <summary>Outlet Clamps</summary>
	XV_03_Right_Retract_Solenoid_Valve							AT %Q*	: BOOL;
    /// <summary>Outlet Clamps</summary>
	XV_03_Right_Extend_Solenoid_Valve							AT %Q*	: BOOL;

	/// <summary>XV-02</summary>
	{attribute 'OPC.UA.DA' := '1'}  				                
	repres_valve														: BOOL;
    /// <summary>XV-02</summary>
	{attribute 'OPC.UA.DA' := '1'}  				                
	{attribute 'OPC.UA.DA.Access' := '1'}  				                
	repres_valve_open_cmd_status										: BOOL;
    /// <summary>XV-02</summary>
	{attribute 'OPC.UA.DA' := '1'}  				                
	{attribute 'OPC.UA.DA.Access' := '1'}  				                
	repres_valve_open											AT %I*	: BOOL;
    /// <summary>XV-02</summary>
	{attribute 'OPC.UA.DA' := '1'}  				                
	{attribute 'OPC.UA.DA.Access' := '1'}  				                
	repres_valve_closed											AT %I*	: BOOL;
    /// <summary>repres valve</summary>
	XV_02														AT %Q*	: BOOL;
	
   /// <summary>01-TT-01</summary>
	{attribute 'OPC.UA.DA' := '1'}  				                
	{attribute 'OPC.UA.DA.Access' := '1'}  				                
	cart01_front_temp													: REAL;
    /// <summary>01-TT-01</summary>
	{attribute 'OPC.UA.DA' := '1'}  				                
	{attribute 'OPC.UA.DA.Access' := '1'}  				                
	cart01_front_temp_error												: BOOL;
    /// <summary>Cart01 front temperature</summary>
	_01_TT_01													AT %I*	: INT;
    /// <summary>Cart01 front temperature</summary>
	_01_TT_01_Error												AT %I*	: BOOL;

    /// <summary>01-TT-03</summary>
	{attribute 'OPC.UA.DA' := '1'}  				                
	{attribute 'OPC.UA.DA.Access' := '1'}  				                
	cart01_back_temp													: REAL;
    /// <summary>01-TT-03</summary>
	{attribute 'OPC.UA.DA' := '1'}  				                
	{attribute 'OPC.UA.DA.Access' := '1'}  				                
	cart01_back_temp_error												: BOOL;
    /// <summary>Cart01 back temperature</summary>
	_01_TT_03													AT %I*	: INT;
    /// <summary>Cart01 back temperature</summary>
	_01_TT_03_Error												AT %I*	: BOOL;
	
    /// <summary>02-TT-01</summary>
	{attribute 'OPC.UA.DA' := '1'}  				                
	{attribute 'OPC.UA.DA.Access' := '1'}  				                
	cart02_front_temp													: REAL;
    /// <summary>02-TT-01</summary>
	{attribute 'OPC.UA.DA' := '1'}  				                
	{attribute 'OPC.UA.DA.Access' := '1'}  				                
	cart02_front_temp_error												: BOOL;
    /// <summary>Cart02 front temperature</summary>
	_02_TT_01													AT %I*	: INT;
    /// <summary>Cart02 front temperature</summary>
	_02_TT_01_Error												AT %I*	: BOOL;

    /// <summary>02-TT-03</summary>
	{attribute 'OPC.UA.DA' := '1'}  				                
	{attribute 'OPC.UA.DA.Access' := '1'}  				                
	cart02_back_temp													: REAL;
    /// <summary>02-TT-03</summary>
	{attribute 'OPC.UA.DA' := '1'}  				                
	{attribute 'OPC.UA.DA.Access' := '1'}  				                
	cart02_back_temp_error												: BOOL;
    /// <summary>Cart02 back temperature</summary>
	_02_TT_03													AT %I*	: INT;
    /// <summary>Cart02 back temperature</summary>
	_02_TT_03_Error												AT %I*	: BOOL;
	
    /// <summary>03-TT-01</summary>
	{attribute 'OPC.UA.DA' := '1'}  				                
	{attribute 'OPC.UA.DA.Access' := '1'}  				                
	cart03_front_temp													: REAL;
    /// <summary>03-TT-01</summary>
	{attribute 'OPC.UA.DA' := '1'}  				                
	{attribute 'OPC.UA.DA.Access' := '1'}  				                
	cart03_front_temp_error												: BOOL;
    /// <summary>Cart03 front temperature</summary>
	_03_TT_01													AT %I*	: INT;
    /// <summary>Cart03 front temperature</summary>
	_03_TT_01_Error												AT %I*	: BOOL;

    /// <summary>03-TT-03</summary>
	{attribute 'OPC.UA.DA' := '1'}  				                
	{attribute 'OPC.UA.DA.Access' := '1'}  				                
	cart03_back_temp													: REAL;
    /// <summary>03-TT-03</summary>
	{attribute 'OPC.UA.DA' := '1'}  				                
	{attribute 'OPC.UA.DA.Access' := '1'}  				                
	cart03_back_temp_error												: BOOL;
    /// <summary>Cart03 back temperature</summary>
	_03_TT_03													AT %I*	: INT;
    /// <summary>Cart03 back temperature</summary>
	_03_TT_03_Error												AT %I*	: BOOL;

    /// <summary>04-TT-01</summary>
	{attribute 'OPC.UA.DA' := '1'}  				                
	{attribute 'OPC.UA.DA.Access' := '1'}  				                
	cart04_front_temp													: REAL;
    /// <summary>04-TT-01</summary>
	{attribute 'OPC.UA.DA' := '1'}  				                
	{attribute 'OPC.UA.DA.Access' := '1'}  				                
	cart04_front_temp_error												: BOOL;
    /// <summary>Cart04 front temperature</summary>
	_04_TT_01													AT %I*	: INT;
    /// <summary>Cart04 front temperature</summary>
	_04_TT_01_Error												AT %I*	: BOOL;

    /// <summary>04-TT-03</summary>
	{attribute 'OPC.UA.DA' := '1'}  				                
	{attribute 'OPC.UA.DA.Access' := '1'}  				                
	cart04_back_temp													: REAL;
    /// <summary>04-TT-03</summary>
	{attribute 'OPC.UA.DA' := '1'}  				                
	{attribute 'OPC.UA.DA.Access' := '1'}  				                
	cart04_back_temp_error												: BOOL;
    /// <summary>Cart04 back temperature</summary>
	_04_TT_03													AT %I*	: INT;
    /// <summary>Cart04 back temperature</summary>
	_04_TT_03_Error												AT %I*	: BOOL;

    /// <summary>05-TT-01</summary>
	{attribute 'OPC.UA.DA' := '1'}  				                
	{attribute 'OPC.UA.DA.Access' := '1'}  				                
	cart05_front_temp													: REAL;
    /// <summary>05-TT-01</summary>
	{attribute 'OPC.UA.DA' := '1'}  				                
	{attribute 'OPC.UA.DA.Access' := '1'}  				                
	cart05_front_temp_error												: BOOL;
    /// <summary>Cart05 front temperature</summary>
	_05_TT_01													AT %I*	: INT;
    /// <summary>Cart05 front temperature</summary>
	_05_TT_01_Error												AT %I*	: BOOL;

    /// <summary>05-TT-03</summary>
	{attribute 'OPC.UA.DA' := '1'}  				                
	{attribute 'OPC.UA.DA.Access' := '1'}  				                
	cart05_back_temp													: REAL;
    /// <summary>05-TT-03</summary>
	{attribute 'OPC.UA.DA' := '1'}  				                
	{attribute 'OPC.UA.DA.Access' := '1'}  				                
	cart05_back_temp_error												: BOOL;
    /// <summary>Cart05 back temperature</summary>
	_05_TT_03													AT %I*	: INT;
    /// <summary>Cart05 back temperature</summary>
	_05_TT_03_Error												AT %I*	: BOOL;
	
    /// <summary>06-TT-01</summary>
	{attribute 'OPC.UA.DA' := '1'}  				                
	{attribute 'OPC.UA.DA.Access' := '1'}  				                
	cart06_front_temp													: REAL;
    /// <summary>06-TT-01</summary>
	{attribute 'OPC.UA.DA' := '1'}  				                
	{attribute 'OPC.UA.DA.Access' := '1'}  				                
	cart06_front_temp_error												: BOOL;
    /// <summary>Cart06 front temperature</summary>
	_06_TT_01													AT %I*	: INT;
    /// <summary>Cart06 front temperature</summary>
	_06_TT_01_Error												AT %I*	: BOOL;

    /// <summary>06-TT-03</summary>
	{attribute 'OPC.UA.DA' := '1'}  				                
	{attribute 'OPC.UA.DA.Access' := '1'}  				                
	cart06_back_temp													: REAL;
    /// <summary>06-TT-03</summary>
	{attribute 'OPC.UA.DA' := '1'}  				                
	{attribute 'OPC.UA.DA.Access' := '1'}  				                
	cart06_back_temp_error												: BOOL;
    /// <summary>Cart06 back temperature</summary>
	_06_TT_03													AT %I*	: INT;
    /// <summary>Cart06 back temperature</summary>
	_06_TT_03_Error												AT %I*	: BOOL;
	
    /// <summary>07-TT-01</summary>
	{attribute 'OPC.UA.DA' := '1'}  				                
	{attribute 'OPC.UA.DA.Access' := '1'}  				                
	cart07_front_temp													: REAL;
    /// <summary>07-TT-01</summary>
	{attribute 'OPC.UA.DA' := '1'}  				                
	{attribute 'OPC.UA.DA.Access' := '1'}  				                
	cart07_front_temp_error												: BOOL;
    /// <summary>Cart07 front temperature</summary>
	_07_TT_01													AT %I*	: INT;
    /// <summary>Cart07 front temperature</summary>
	_07_TT_01_Error												AT %I*	: BOOL;

    /// <summary>07-TT-03</summary>
	{attribute 'OPC.UA.DA' := '1'}  				                
	{attribute 'OPC.UA.DA.Access' := '1'}  				                
	cart07_back_temp													: REAL;
    /// <summary>07-TT-03</summary>
	{attribute 'OPC.UA.DA' := '1'}  				                
	{attribute 'OPC.UA.DA.Access' := '1'}  				                
	cart07_back_temp_error												: BOOL;
    /// <summary>Cart07 back temperature</summary>
	_07_TT_03													AT %I*	: INT;
    /// <summary>Cart07 back temperature</summary>
	_07_TT_03_Error												AT %I*	: BOOL;
	
    /// <summary>08-TT-01</summary>
	{attribute 'OPC.UA.DA' := '1'}  				                
	{attribute 'OPC.UA.DA.Access' := '1'}  				                
	cart08_front_temp													: REAL;
    /// <summary>08-TT-01</summary>
	{attribute 'OPC.UA.DA' := '1'}  				                
	{attribute 'OPC.UA.DA.Access' := '1'}  				                
	cart08_front_temp_error												: BOOL;
    /// <summary>Cart08 front temperature</summary>
	_08_TT_01													AT %I*	: INT;
    /// <summary>Cart08 front temperature</summary>
	_08_TT_01_Error												AT %I*	: BOOL;

    /// <summary>08-TT-03</summary>
	{attribute 'OPC.UA.DA' := '1'}  				                
	{attribute 'OPC.UA.DA.Access' := '1'}  				                
	cart08_back_temp													: REAL;
    /// <summary>08-TT-03</summary>
	{attribute 'OPC.UA.DA' := '1'}  				                
	{attribute 'OPC.UA.DA.Access' := '1'}  				                
	cart08_back_temp_error												: BOOL;
    /// <summary>Cart08 back temperature</summary>
	_08_TT_03													AT %I*	: INT;
    /// <summary>Cart08 back temperature</summary>
	_08_TT_03_Error												AT %I*	: BOOL;
	
    /// <summary>09-TT-01</summary>
	{attribute 'OPC.UA.DA' := '1'}  				                
	{attribute 'OPC.UA.DA.Access' := '1'}  				                
	cart09_front_temp													: REAL;
    /// <summary>09-TT-01</summary>
	{attribute 'OPC.UA.DA' := '1'}  				                
	{attribute 'OPC.UA.DA.Access' := '1'}  				                
	cart09_front_temp_error												: BOOL;
    /// <summary>Cart09 front temperature</summary>
	_09_TT_01													AT %I*	: INT;
    /// <summary>Cart09 front temperature</summary>
	_09_TT_01_Error												AT %I*	: BOOL;

    /// <summary>09-TT-03</summary>
	{attribute 'OPC.UA.DA' := '1'}  				                
	{attribute 'OPC.UA.DA.Access' := '1'}  				                
	cart09_back_temp													: REAL;
    /// <summary>09-TT-03</summary>
	{attribute 'OPC.UA.DA' := '1'}  				                
	{attribute 'OPC.UA.DA.Access' := '1'}  				                
	cart09_back_temp_error												: BOOL;
    /// <summary>Cart09 back temperature</summary>
	_09_TT_03													AT %I*	: INT;
    /// <summary>Cart09 back temperature</summary>
	_09_TT_03_Error												AT %I*	: BOOL;
	
    /// <summary>10-TT-01</summary>
	{attribute 'OPC.UA.DA' := '1'}  				                
	{attribute 'OPC.UA.DA.Access' := '1'}  				                
	cart10_front_temp													: REAL;
    /// <summary>10-TT-01</summary>
	{attribute 'OPC.UA.DA' := '1'}  				                
	{attribute 'OPC.UA.DA.Access' := '1'}  				                
	cart10_front_temp_error												: BOOL;
    /// <summary>Cart10 front temperature</summary>
	_10_TT_01													AT %I*	: INT;
    /// <summary>Cart10 front temperature</summary>
	_10_TT_01_Error												AT %I*	: BOOL;

    /// <summary>10-TT-03</summary>
	{attribute 'OPC.UA.DA' := '1'}  				                
	{attribute 'OPC.UA.DA.Access' := '1'}  				                
	cart10_back_temp													: REAL;
    /// <summary>10-TT-03</summary>
	{attribute 'OPC.UA.DA' := '1'}  				                
	{attribute 'OPC.UA.DA.Access' := '1'}  				                
	cart10_back_temp_error												: BOOL;
    /// <summary>Cart10 back temperature</summary>
	_10_TT_03													AT %I*	: INT;
    /// <summary>Cart10 back temperature</summary>
	_10_TT_03_Error												AT %I*	: BOOL;

    /// <summary>11-TT-01</summary>
	{attribute 'OPC.UA.DA' := '1'}  				                
	{attribute 'OPC.UA.DA.Access' := '1'}  				                
	cart11_front_temp													: REAL;
    /// <summary>11-TT-01</summary>
	{attribute 'OPC.UA.DA' := '1'}  				                
	{attribute 'OPC.UA.DA.Access' := '1'}  				                
	cart11_front_temp_error												: BOOL;
    /// <summary>Cart11 front temperature</summary>
	_11_TT_01													AT %I*	: INT;
    /// <summary>Cart11 front temperature</summary>
	_11_TT_01_Error												AT %I*	: BOOL;

    /// <summary>11-TT-03</summary>
	{attribute 'OPC.UA.DA' := '1'}  				                
	{attribute 'OPC.UA.DA.Access' := '1'}  				                
	cart11_back_temp													: REAL;
    /// <summary>11-TT-03</summary>
	{attribute 'OPC.UA.DA' := '1'}  				                
	{attribute 'OPC.UA.DA.Access' := '1'}  				                
	cart11_back_temp_error												: BOOL;
    /// <summary>Cart11 back temperature</summary>
	_11_TT_03													AT %I*	: INT;
    /// <summary>Cart11 back temperature</summary>
	_11_TT_03_Error												AT %I*	: BOOL;

    /// <summary>12-TT-01</summary>
	{attribute 'OPC.UA.DA' := '1'}  				                
	{attribute 'OPC.UA.DA.Access' := '1'}  				                
	cart12_front_temp													: REAL;
    /// <summary>12-TT-01</summary>
	{attribute 'OPC.UA.DA' := '1'}  				                
	{attribute 'OPC.UA.DA.Access' := '1'}  				                
	cart12_front_temp_error												: BOOL;
    /// <summary>Cart12 front temperature</summary>
	_12_TT_01													AT %I*	: INT;
    /// <summary>Cart12 front temperature</summary>
	_12_TT_01_Error												AT %I*	: BOOL;

    /// <summary>12-TT-03</summary>
	{attribute 'OPC.UA.DA' := '1'}  				                
	{attribute 'OPC.UA.DA.Access' := '1'}  				                
	cart12_back_temp													: REAL;
    /// <summary>12-TT-03</summary>
	{attribute 'OPC.UA.DA' := '1'}  				                
	{attribute 'OPC.UA.DA.Access' := '1'}  				                
	cart12_back_temp_error												: BOOL;
    /// <summary>Cart12 back temperature</summary>
	_12_TT_03													AT %I*	: INT;
    /// <summary>Cart12 back temperature</summary>
	_12_TT_03_Error												AT %I*	: BOOL;
	
	{attribute 'OPC.UA.DA' := '1'}  				                
	{attribute 'OPC.UA.DA.Access' := '1'}  				                
	temp_low															: REAL;
	{attribute 'OPC.UA.DA' := '1'}  				                
	{attribute 'OPC.UA.DA.Access' := '1'}  				                
	temp_high															: REAL;
	{attribute 'OPC.UA.DA' := '1'}  				                
	{attribute 'OPC.UA.DA.Access' := '1'}  				                
	temp_average														: REAL;

	desorption_air_high_temp_count										: INT;
	adsorption_high_temp_count											: INT;
	vacuum_cooling_high_temp_count										: INT;

END_VAR

VAR_GLOBAL PERSISTENT

    /// <summary>AT-01</summary>
	{attribute 'OPC.UA.DA' := '1'}  				                
	inlet_co2_low														: REAL;							// Tag for low point to scale input (these tags can be preset as shown or overwritten)
    /// <summary>AT-01</summary>
	{attribute 'OPC.UA.DA' := '1'}  				                
	inlet_co2_high														: REAL;							// Tag for high point to scale input
    /// <summary>AT-01</summary>
	{attribute 'OPC.UA.DA' := '1'}  				                
	inlet_co2_min														: REAL;							// Tag for minimum display value (if input is below this value, zero is displayed)
    /// <summary>AT-01</summary>
	{attribute 'OPC.UA.DA' := '1'}  				                
	inlet_co2_offset													: REAL;							// Tag for offset correction value

    /// <summary>AT-02</summary>
	{attribute 'OPC.UA.DA' := '1'}  				                
	inlet_h2o_low														: REAL;
    /// <summary>AT-02</summary>
	{attribute 'OPC.UA.DA' := '1'}  				                
	inlet_h2o_high														: REAL;
    /// <summary>AT-02</summary>
	{attribute 'OPC.UA.DA' := '1'}  				                
	inlet_h2o_min														: REAL;
    /// <summary>AT-02</summary>
	{attribute 'OPC.UA.DA' := '1'}  				                
	inlet_h2o_offset													: REAL;

    /// <summary>AT-03</summary>
	{attribute 'OPC.UA.DA' := '1'}  				                
	outlet_co2_low														: REAL;
    /// <summary>AT-03</summary>
	{attribute 'OPC.UA.DA' := '1'}  				                
	outlet_co2_high														: REAL;
    /// <summary>AT-03</summary>
	{attribute 'OPC.UA.DA' := '1'}  				                
	outlet_co2_min														: REAL;
    /// <summary>AT-03</summary>
	{attribute 'OPC.UA.DA' := '1'}  				                
	outlet_co2_offset													: REAL;

    /// <summary>AT-04</summary>
	{attribute 'OPC.UA.DA' := '1'}  				                
	outlet_h2o_low														: REAL;
    /// <summary>AT-04</summary>
	{attribute 'OPC.UA.DA' := '1'}  				                
	outlet_h2o_high														: REAL;
    /// <summary>AT-04</summary>
	{attribute 'OPC.UA.DA' := '1'}  				                
	outlet_h2o_min														: REAL;
    /// <summary>AT-04</summary>
	{attribute 'OPC.UA.DA' := '1'}  				                
	outlet_h2o_offset													: REAL;
	
    /// <summary>FT-01</summary>
	{attribute 'OPC.UA.DA' := '1'}  				                
	air_flow_low														: REAL;
    /// <summary>FT-01</summary>
	{attribute 'OPC.UA.DA' := '1'}  				                
	air_flow_high														: REAL;
    /// <summary>FT-01</summary>
	{attribute 'OPC.UA.DA' := '1'}  				                
	air_flow_min														: REAL;
    /// <summary>FT-01</summary>
	{attribute 'OPC.UA.DA' := '1'}  				                
	air_flow_offset														: REAL;

    /// <summary>PDT-01</summary>
	{attribute 'OPC.UA.DA' := '1'}  				                
	filter_diff_pres_low												: REAL;
    /// <summary>PDT-01</summary>
	{attribute 'OPC.UA.DA' := '1'}  				                
	filter_diff_pres_high												: REAL;
    /// <summary>PDT-01</summary>
	{attribute 'OPC.UA.DA' := '1'}  				                
	filter_diff_pres_min												: REAL;
    /// <summary>PDT-01</summary>
	{attribute 'OPC.UA.DA' := '1'}  				                
	filter_diff_pres_offset												: REAL;

    /// <summary>PDT-02</summary>
	{attribute 'OPC.UA.DA' := '1'}  				                
	sorbent_diff_pres_low												: REAL;
    /// <summary>PDT-02</summary>
	{attribute 'OPC.UA.DA' := '1'}  				                
	sorbent_diff_pres_high												: REAL;
    /// <summary>PDT-02</summary>
	{attribute 'OPC.UA.DA' := '1'}  				                
	sorbent_diff_pres_min												: REAL;
    /// <summary>PDT-02</summary>
	{attribute 'OPC.UA.DA' := '1'}  				                
	sorbent_diff_pres_offset											: REAL;

    /// <summary>PDT-03</summary>
	{attribute 'OPC.UA.DA' := '1'}  				                
	fan_diff_pres_low													: REAL;
    /// <summary>PDT-03</summary>
	{attribute 'OPC.UA.DA' := '1'}  				                
	fan_diff_pres_high													: REAL;
    /// <summary>PDT-03</summary>
	{attribute 'OPC.UA.DA' := '1'}  				                
	fan_diff_pres_min													: REAL;
    /// <summary>PDT-03</summary>
	{attribute 'OPC.UA.DA' := '1'}  				                
	fan_diff_pres_offset												: REAL;

    /// <summary>PT-01</summary>
	{attribute 'OPC.UA.DA' := '1'}  				                
	reactor_pres_low													: REAL;
    /// <summary>PT-01</summary>
	{attribute 'OPC.UA.DA' := '1'}  				                
	reactor_pres_high													: REAL;
    /// <summary>PT-01</summary>
	{attribute 'OPC.UA.DA' := '1'}  				                
	reactor_pres_min													: REAL;
    /// <summary>PT-01</summary>
	{attribute 'OPC.UA.DA' := '1'}  				                
	reactor_pres_offset													: REAL;

    /// <summary>TT-05</summary>
	{attribute 'OPC.UA.DA' := '1'}  				                
	reactor_wall_temp_offset											: REAL;

    /// <summary>TT-06</summary>
	{attribute 'OPC.UA.DA' := '1'}  				                
	outlet_line_temp_offset												: REAL;

	
    /// <summary>01-TT-01</summary>
	{attribute 'OPC.UA.DA' := '1'}  				                
	cart01_front_temp_offset											: REAL;
    /// <summary>10-TT-03</summary>
	{attribute 'OPC.UA.DA' := '1'}  				                
	cart01_back_temp_offset												: REAL;
    /// <summary>02-TT-01</summary>
	{attribute 'OPC.UA.DA' := '1'}  				                
	cart02_front_temp_offset											: REAL;
    /// <summary>02-TT-03</summary>
	{attribute 'OPC.UA.DA' := '1'}  				                
	cart02_back_temp_offset												: REAL;
    /// <summary>03-TT-01</summary>
	{attribute 'OPC.UA.DA' := '1'}  				                
	cart03_front_temp_offset											: REAL;
    /// <summary>03-TT-03</summary>
	{attribute 'OPC.UA.DA' := '1'}  				                
	cart03_back_temp_offset												: REAL;
    /// <summary>04-TT-01</summary>
	{attribute 'OPC.UA.DA' := '1'}  				                
	cart04_front_temp_offset											: REAL;
    /// <summary>04-TT-03</summary>
	{attribute 'OPC.UA.DA' := '1'}  				                
	cart04_back_temp_offset												: REAL;
    /// <summary>05-TT-01</summary>
	{attribute 'OPC.UA.DA' := '1'}  				                
	cart05_front_temp_offset											: REAL;
    /// <summary>05-TT-03</summary>
	{attribute 'OPC.UA.DA' := '1'}  				                
	cart05_back_temp_offset												: REAL;
    /// <summary>06-TT-01</summary>
	{attribute 'OPC.UA.DA' := '1'}  				                
	cart06_front_temp_offset											: REAL;
    /// <summary>06-TT-03</summary>
	{attribute 'OPC.UA.DA' := '1'}  				                
	cart06_back_temp_offset												: REAL;
    /// <summary>07-TT-01</summary>
	{attribute 'OPC.UA.DA' := '1'}  				                
	cart07_front_temp_offset											: REAL;
    /// <summary>07-TT-03</summary>
	{attribute 'OPC.UA.DA' := '1'}  				                
	cart07_back_temp_offset												: REAL;
    /// <summary>08-TT-01</summary>
	{attribute 'OPC.UA.DA' := '1'}  				                
	cart08_front_temp_offset											: REAL;
    /// <summary>08-TT-03</summary>
	{attribute 'OPC.UA.DA' := '1'}  				                
	cart08_back_temp_offset												: REAL;
    /// <summary>09-TT-01</summary>
	{attribute 'OPC.UA.DA' := '1'}  				                
	cart09_front_temp_offset											: REAL;
    /// <summary>09-TT-03</summary>
	{attribute 'OPC.UA.DA' := '1'}  				                
	cart09_back_temp_offset												: REAL;
    /// <summary>10-TT-01</summary>
	{attribute 'OPC.UA.DA' := '1'}  				                
	cart10_front_temp_offset											: REAL;
    /// <summary>10-TT-03</summary>
	{attribute 'OPC.UA.DA' := '1'}  				                
	cart10_back_temp_offset												: REAL;
    /// <summary>11-TT-01</summary>
	{attribute 'OPC.UA.DA' := '1'}  				                
	cart11_front_temp_offset											: REAL;
    /// <summary>11-TT-03</summary>
	{attribute 'OPC.UA.DA' := '1'}  				                
	cart11_back_temp_offset												: REAL;
    /// <summary>12-TT-01</summary>
	{attribute 'OPC.UA.DA' := '1'}  				                
	cart12_front_temp_offset											: REAL;
    /// <summary>12-TT-03</summary>
	{attribute 'OPC.UA.DA' := '1'}  				                
	cart12_back_temp_offset												: REAL;
	
END_VAR

// ---- GVLs/m01_rs2.TcGVL
// Phase 0 - m01_rs2
// Rev 1.0 - April 24, 2024

{attribute 'qualified_only'}
VAR_GLOBAL
 
	{attribute 'OPC.UA.DA' := '1'}  				                
	{attribute 'OPC.UA.DA.Access' := '1'}  				                
	ti_Total_Cycle_Count												: DINT; 
	{attribute 'OPC.UA.DA' := '1'}  				                
	{attribute 'OPC.UA.DA.Access' := '1'}  				                
	ti_Cycle_Count														: INT; 
	{attribute 'OPC.UA.DA' := '1'}  				                
	{attribute 'OPC.UA.DA.Access' := '1'}  				                
	ti_Machine_State													: INT;
	{attribute 'OPC.UA.DA' := '1'}  				                
	{attribute 'OPC.UA.DA.Access' := '1'}  				                
	ti_Current_Step														: INT;
	{attribute 'OPC.UA.DA' := '1'}  				                
	{attribute 'OPC.UA.DA.Access' := '1'}  				                
	tb_Process_Running													: BOOL;
	{attribute 'OPC.UA.DA' := '1'}  				                
	{attribute 'OPC.UA.DA.Access' := '1'}  				                
	tb_Repressurization_Running											: BOOL;
	{attribute 'OPC.UA.DA' := '1'}  				                
	{attribute 'OPC.UA.DA.Access' := '1'}  				                
	tb_Adsorption_Running												: BOOL;
	{attribute 'OPC.UA.DA' := '1'}  				                
	{attribute 'OPC.UA.DA.Access' := '1'}  				                
	tb_Evacuation_Running												: BOOL;
	{attribute 'OPC.UA.DA' := '1'}  				                
	{attribute 'OPC.UA.DA.Access' := '1'}  				                
	tb_Desorption_Running												: BOOL;
	{attribute 'OPC.UA.DA' := '1'}  				                
	{attribute 'OPC.UA.DA.Access' := '1'}  				                
	tb_Process_Complete													: BOOL;
	{attribute 'OPC.UA.DA' := '1'}  				                
	{attribute 'OPC.UA.DA.Access' := '1'}  				                
	tr_Remaining_Time													: REAL;
	{attribute 'OPC.UA.DA' := '1'}  				                
	{attribute 'OPC.UA.DA.Access' := '1'}  				                
	ti_Status															: INT;
	{attribute 'OPC.UA.DA' := '1'}  				                
	{attribute 'OPC.UA.DA.Access' := '1'}  				                
	ts_Status_Text														: STRING;		

	
	{attribute 'OPC.UA.DA' := '1'}  				                
	{attribute 'OPC.UA.DA.Access' := '1'}  				                
	cycle_stage															: STRING;


    /// <summary>PWR-01</summary>
	{attribute 'OPC.UA.DA' := '1'}  				                
	power_control														: BOOL;
    /// <summary>PWR-01</summary>
	{attribute 'OPC.UA.DA' := '1'}  				                
	{attribute 'OPC.UA.DA.Access' := '1'}  				                
	power_control_status												: BOOL;
    /// <summary>power_cmd</summary>
	PWR_01														AT %Q*	: BOOL;
	circuit_breaker_no_feedback									AT %I*	: BOOL;
	circuit_breaker_nc_feedback									AT %I*	: BOOL;
	
    /// <summary>LS-01</summary>
	{attribute 'OPC.UA.DA' := '1'}  				                
	{attribute 'OPC.UA.DA.Access' := '1'}  				                
	condensate_lsl												AT %I*	: BOOL;
	
    /// <summary>LS-02</summary>
	{attribute 'OPC.UA.DA' := '1'}  				                
	{attribute 'OPC.UA.DA.Access' := '1'}  				                
	condensate_lsh												AT %I*	: BOOL;

    /// <summary>P-01</summary>
	{attribute 'OPC.UA.DA' := '1'}  				                
	condensate_pump														: BOOL;
    /// <summary>P-01</summary>
	{attribute 'OPC.UA.DA' := '1'}  				                
	{attribute 'OPC.UA.DA.Access' := '1'}  				                
	condensate_pump_cmd_status											: BOOL;
    /// <summary>condensate pump</summary>
	P_01														AT %Q*	: BOOL;

    /// <summary>PCV-01</summary>
	{attribute 'OPC.UA.DA' := '1'}  				                
	steam_control_valve													: REAL;
    /// <summary>PCV-01</summary>
	{attribute 'OPC.UA.DA' := '1'}  				                
	{attribute 'OPC.UA.DA.Access' := '1'}  				                
	steam_control_valve_position										: REAL;
    /// <summary>steam control valve</summary>
	PCV_01														AT %Q*	: INT;
    /// <summary>steam control valve</summary>
	PCV_01_position												AT %I*	: INT;
    /// <summary>PCV-01</summary>
	{attribute 'OPC.UA.DA' := '1'}  				                
	{attribute 'OPC.UA.DA.Access' := '1'}  				                
	steam_control_valve_position_error							AT %I*	: BOOL;
    /// <summary>PCV-01</summary>                  	           
	{attribute 'OPC.UA.DA' := '1'}  				                
	steam_control_valve_mode											: INT;			
    /// <summary>PCV-01</summary>                  	           
	{attribute 'OPC.UA.DA' := '1'}  				                
	{attribute 'OPC.UA.DA.Access' := '1'}  				                
	steam_control_valve_current_mode									: INT;			
    /// <summary>PCV-01</summary>                  	           
	steam_control_valve_kp												: REAL		:= 0.01; 
    /// <summary>PCV-01</summary>                  	           
	steam_control_valve_ki												: REAL		:= 0.01;
    /// <summary>PCV-01</summary>                  	           
	steam_control_valve_loop_time										: REAL		:= 2000;
    /// <summary>PCV-01</summary>                  	           
	steam_control_valve_iband											: REAL		:= 6;
    /// <summary>PCV-01</summary>                  	           
	steam_control_valve_base											: INT		:= 13110;
    /// <summary>PCV-01</summary>                  	           
	steam_control_valve_base_adjust										: INT		:= 10;
		                                	        	
    /// <summary>XV-04</summary>
	{attribute 'OPC.UA.DA' := '1'}  				                
	dead_air_valve														: BOOL;
    /// <summary>XV-04</summary>
	{attribute 'OPC.UA.DA' := '1'}  				                
	{attribute 'OPC.UA.DA.Access' := '1'}  				                
	dead_air_valve_open_cmd_status										: BOOL;
    /// <summary>XV-04</summary>
	{attribute 'OPC.UA.DA' := '1'}  				                
	{attribute 'OPC.UA.DA.Access' := '1'}  				                
	dead_air_valve_open											AT %I*	: BOOL;
    /// <summary>XV-04</summary>
	{attribute 'OPC.UA.DA' := '1'}  				                
	{attribute 'OPC.UA.DA.Access' := '1'}  				                
	dead_air_valve_closed										AT %I*	: BOOL;
    /// <summary>dead air valve</summary>
	XV_04														AT %Q*	: BOOL;
	
    /// <summary>XV-05</summary>
	{attribute 'OPC.UA.DA' := '1'}  				                
	purge_valve															: BOOL;
    /// <summary>XV-05</summary>
	{attribute 'OPC.UA.DA' := '1'}  				                
	{attribute 'OPC.UA.DA.Access' := '1'}  				                
	purge_valve_open_cmd_status											: BOOL;
    /// <summary>XV-05</summary>
	{attribute 'OPC.UA.DA' := '1'}  				                
	{attribute 'OPC.UA.DA.Access' := '1'}  				                
	purge_valve_open											AT %I*	: BOOL;
    /// <summary>XV-05</summary>
	{attribute 'OPC.UA.DA' := '1'}  				                
	{attribute 'OPC.UA.DA.Access' := '1'}  				                
	purge_valve_closed											AT %I*	: BOOL;
    /// <summary>purge valve</summary>
	XV_05														AT %Q*	: BOOL;
	
    /// <summary>XV-06</summary>
	{attribute 'OPC.UA.DA' := '1'}  				                
	cooling_valve														: BOOL;
    /// <summary>XV-06</summary>
	{attribute 'OPC.UA.DA' := '1'}  				                
	{attribute 'OPC.UA.DA.Access' := '1'}  				                
	cooling_valve_open_cmd_status										: BOOL;
    /// <summary>XV-06</summary>
	{attribute 'OPC.UA.DA' := '1'}  				                
	{attribute 'OPC.UA.DA.Access' := '1'}  				                
	cooling_valve_open											AT %I*	: BOOL;
    /// <summary>XV-06</summary>
	{attribute 'OPC.UA.DA' := '1'}  				                
	{attribute 'OPC.UA.DA.Access' := '1'}  				                
	cooling_valve_closed										AT %I*	: BOOL;
    /// <summary>cooling valve</summary>
	XV_06														AT %Q*	: BOOL;
	
    /// <summary>XV-07</summary>
	{attribute 'OPC.UA.DA' := '1'}  				                
	steam_header_valve													: BOOL;
    /// <summary>XV-07</summary>
	{attribute 'OPC.UA.DA' := '1'}  				                
	{attribute 'OPC.UA.DA.Access' := '1'}  				                
	steam_header_valve_open_cmd_status									: BOOL;
    /// <summary>XV-07</summary>
	{attribute 'OPC.UA.DA' := '1'}  				                
	{attribute 'OPC.UA.DA.Access' := '1'}  				                
	steam_header_valve_open										AT %I*	: BOOL;
    /// <summary>XV-07</summary>
	{attribute 'OPC.UA.DA' := '1'}  				                
	{attribute 'OPC.UA.DA.Access' := '1'}  				                
	steam_header_valve_closed									AT %I*	: BOOL;
    /// <summary>steam header valve</summary>
	XV_07														AT %Q*	: BOOL;

END_VAR

// ---- GVLs/m01_rs3.TcGVL
// Phase 0 - m01_rs3
// Rev 1.0 - April 24, 2024

{attribute 'qualified_only'}
VAR_GLOBAL
 
	{attribute 'OPC.UA.DA' := '1'}  				                
	{attribute 'OPC.UA.DA.Access' := '1'}  				                
	ti_Total_Cycle_Count												: DINT; 
	{attribute 'OPC.UA.DA' := '1'}  				                
	{attribute 'OPC.UA.DA.Access' := '1'}  				                
	ti_Cycle_Count														: INT; 
	{attribute 'OPC.UA.DA' := '1'}  				                
	{attribute 'OPC.UA.DA.Access' := '1'}  				                
	ti_Machine_State													: INT;
	{attribute 'OPC.UA.DA' := '1'}  				                
	{attribute 'OPC.UA.DA.Access' := '1'}  				                
	ti_Current_Step														: INT;
	{attribute 'OPC.UA.DA' := '1'}  				                
	{attribute 'OPC.UA.DA.Access' := '1'}  				                
	tb_Process_Running													: BOOL;
	{attribute 'OPC.UA.DA' := '1'}  				                
	{attribute 'OPC.UA.DA.Access' := '1'}  				                
	tb_Repressurization_Running											: BOOL;
	{attribute 'OPC.UA.DA' := '1'}  				                
	{attribute 'OPC.UA.DA.Access' := '1'}  				                
	tb_Adsorption_Running												: BOOL;
	{attribute 'OPC.UA.DA' := '1'}  				                
	{attribute 'OPC.UA.DA.Access' := '1'}  				                
	tb_Evacuation_Running												: BOOL;
	{attribute 'OPC.UA.DA' := '1'}  				                
	{attribute 'OPC.UA.DA.Access' := '1'}  				                
	tb_Desorption_Running												: BOOL;
	{attribute 'OPC.UA.DA' := '1'}  				                
	{attribute 'OPC.UA.DA.Access' := '1'}  				                
	tb_Process_Complete													: BOOL;
	{attribute 'OPC.UA.DA' := '1'}  				                
	{attribute 'OPC.UA.DA.Access' := '1'}  				                
	tr_Remaining_Time													: REAL;
	{attribute 'OPC.UA.DA' := '1'}  				                
	{attribute 'OPC.UA.DA.Access' := '1'}  				                
	ti_Status															: INT;
	{attribute 'OPC.UA.DA' := '1'}  				                
	{attribute 'OPC.UA.DA.Access' := '1'}  				                
	ts_Status_Text														: STRING;		

	
	{attribute 'OPC.UA.DA' := '1'}  				                
	{attribute 'OPC.UA.DA.Access' := '1'}  				                
	cycle_stage															: STRING;


    /// <summary>PWR-01</summary>
	{attribute 'OPC.UA.DA' := '1'}  				                
	power_control														: BOOL;
    /// <summary>PWR-01</summary>
	{attribute 'OPC.UA.DA' := '1'}  				                
	{attribute 'OPC.UA.DA.Access' := '1'}  				                
	power_control_status												: BOOL;
    /// <summary>power_cmd</summary>
	PWR_01														AT %Q*	: BOOL;
	circuit_breaker_no_feedback									AT %I*	: BOOL;
	circuit_breaker_nc_feedback									AT %I*	: BOOL;
	
    /// <summary>LS-01</summary>
	{attribute 'OPC.UA.DA' := '1'}  				                
	{attribute 'OPC.UA.DA.Access' := '1'}  				                
	condensate_lsl												AT %I*	: BOOL;
	
    /// <summary>LS-02</summary>
	{attribute 'OPC.UA.DA' := '1'}  				                
	{attribute 'OPC.UA.DA.Access' := '1'}  				                
	condensate_lsh												AT %I*	: BOOL;

    /// <summary>P-01</summary>
	{attribute 'OPC.UA.DA' := '1'}  				                
	condensate_pump														: BOOL;
    /// <summary>P-01</summary>
	{attribute 'OPC.UA.DA' := '1'}  				                
	{attribute 'OPC.UA.DA.Access' := '1'}  				                
	condensate_pump_cmd_status											: BOOL;
    /// <summary>condensate pump</summary>
	P_01														AT %Q*	: BOOL;

    /// <summary>PCV-01</summary>
	{attribute 'OPC.UA.DA' := '1'}  				                
	steam_control_valve													: REAL;
    /// <summary>PCV-01</summary>
	{attribute 'OPC.UA.DA' := '1'}  				                
	{attribute 'OPC.UA.DA.Access' := '1'}  				                
	steam_control_valve_position										: REAL;
    /// <summary>steam control valve</summary>
	PCV_01														AT %Q*	: INT;
    /// <summary>steam control valve</summary>
	PCV_01_position												AT %I*	: INT;
    /// <summary>PCV-01</summary>
	{attribute 'OPC.UA.DA' := '1'}  				                
	{attribute 'OPC.UA.DA.Access' := '1'}  				                
	steam_control_valve_position_error							AT %I*	: BOOL;
    /// <summary>PCV-01</summary>                  	           
	{attribute 'OPC.UA.DA' := '1'}  				                
	steam_control_valve_mode											: INT;			
    /// <summary>PCV-01</summary>                  	           
	{attribute 'OPC.UA.DA' := '1'}  				                
	{attribute 'OPC.UA.DA.Access' := '1'}  				                
	steam_control_valve_current_mode									: INT;			
    /// <summary>PCV-01</summary>                  	           
	steam_control_valve_kp												: REAL		:= 0.01; 
    /// <summary>PCV-01</summary>                  	           
	steam_control_valve_ki												: REAL		:= 0.01;
    /// <summary>PCV-01</summary>                  	           
	steam_control_valve_loop_time										: REAL		:= 2000;
    /// <summary>PCV-01</summary>                  	           
	steam_control_valve_iband											: REAL		:= 6;
    /// <summary>PCV-01</summary>                  	           
	steam_control_valve_base											: INT		:= 13110;
    /// <summary>PCV-01</summary>                  	           
	steam_control_valve_base_adjust										: INT		:= 10;
		                                	        	
    /// <summary>XV-04</summary>
	{attribute 'OPC.UA.DA' := '1'}  				                
	dead_air_valve														: BOOL;
    /// <summary>XV-04</summary>
	{attribute 'OPC.UA.DA' := '1'}  				                
	{attribute 'OPC.UA.DA.Access' := '1'}  				                
	dead_air_valve_open_cmd_status										: BOOL;
    /// <summary>XV-04</summary>
	{attribute 'OPC.UA.DA' := '1'}  				                
	{attribute 'OPC.UA.DA.Access' := '1'}  				                
	dead_air_valve_open											AT %I*	: BOOL;
    /// <summary>XV-04</summary>
	{attribute 'OPC.UA.DA' := '1'}  				                
	{attribute 'OPC.UA.DA.Access' := '1'}  				                
	dead_air_valve_closed										AT %I*	: BOOL;
    /// <summary>dead air valve</summary>
	XV_04														AT %Q*	: BOOL;
	
    /// <summary>XV-05</summary>
	{attribute 'OPC.UA.DA' := '1'}  				                
	purge_valve															: BOOL;
    /// <summary>XV-05</summary>
	{attribute 'OPC.UA.DA' := '1'}  				                
	{attribute 'OPC.UA.DA.Access' := '1'}  				                
	purge_valve_open_cmd_status											: BOOL;
    /// <summary>XV-05</summary>
	{attribute 'OPC.UA.DA' := '1'}  				                
	{attribute 'OPC.UA.DA.Access' := '1'}  				                
	purge_valve_open											AT %I*	: BOOL;
    /// <summary>XV-05</summary>
	{attribute 'OPC.UA.DA' := '1'}  				                
	{attribute 'OPC.UA.DA.Access' := '1'}  				                
	purge_valve_closed											AT %I*	: BOOL;
    /// <summary>purge valve</summary>
	XV_05														AT %Q*	: BOOL;
	
    /// <summary>XV-06</summary>
	{attribute 'OPC.UA.DA' := '1'}  				                
	cooling_valve														: BOOL;
    /// <summary>XV-06</summary>
	{attribute 'OPC.UA.DA' := '1'}  				                
	{attribute 'OPC.UA.DA.Access' := '1'}  				                
	cooling_valve_open_cmd_status										: BOOL;
    /// <summary>XV-06</summary>
	{attribute 'OPC.UA.DA' := '1'}  				                
	{attribute 'OPC.UA.DA.Access' := '1'}  				                
	cooling_valve_open											AT %I*	: BOOL;
    /// <summary>XV-06</summary>
	{attribute 'OPC.UA.DA' := '1'}  				                
	{attribute 'OPC.UA.DA.Access' := '1'}  				                
	cooling_valve_closed										AT %I*	: BOOL;
    /// <summary>cooling valve</summary>
	XV_06														AT %Q*	: BOOL;
	
    /// <summary>XV-07</summary>
	{attribute 'OPC.UA.DA' := '1'}  				                
	steam_header_valve													: BOOL;
    /// <summary>XV-07</summary>
	{attribute 'OPC.UA.DA' := '1'}  				                
	{attribute 'OPC.UA.DA.Access' := '1'}  				                
	steam_header_valve_open_cmd_status									: BOOL;
    /// <summary>XV-07</summary>
	{attribute 'OPC.UA.DA' := '1'}  				                
	{attribute 'OPC.UA.DA.Access' := '1'}  				                
	steam_header_valve_open										AT %I*	: BOOL;
    /// <summary>XV-07</summary>
	{attribute 'OPC.UA.DA' := '1'}  				                
	{attribute 'OPC.UA.DA.Access' := '1'}  				                
	steam_header_valve_closed									AT %I*	: BOOL;
    /// <summary>steam header valve</summary>
	XV_07														AT %Q*	: BOOL;

END_VAR

// ---- GVLs/u01.TcGVL
// Phase 0 - u01
// Rev 1.0 - June 3, 2024

{attribute 'qualified_only'}
VAR_GLOBAL

	AT03_Power												AT %Q*		: BOOL;
	FT02_Power												AT %Q*		: BOOL;
	AT04_06_Power											AT %Q*		: BOOL;
	
	
	shutdown_process													: BOOL;
	{attribute 'OPC.UA.DA' := '1'}  				                
	{attribute 'OPC.UA.DA.Access' := '1'}  				                
	warmup_complete														: BOOL;
	{attribute 'OPC.UA.DA' := '1'}  				                
	{attribute 'OPC.UA.DA.Access' := '1'}  				                
	steam_bypass_complete												: BOOL;

	{attribute 'OPC.UA.DA' := '1'}  				                
	write_persistent_data												: BOOL;
	{attribute 'OPC.UA.DA' := '1'}  				                
	drainage_function_on_or												: BOOL;
	{attribute 'OPC.UA.DA' := '1'}  				                
	drainage_function_off_or											: BOOL;
	{attribute 'OPC.UA.DA' := '1'}  				                
	{attribute 'OPC.UA.DA.Access' := '1'}  				                
	drainage_on															: BOOL;
	
    /// <summary>LS-01</summary>
	{attribute 'OPC.UA.DA' := '1'}  				                
	{attribute 'OPC.UA.DA.Access' := '1'}  				                
	product_condensate_drum_lsl									AT %I*	: BOOL;
    /// <summary>LS-02</summary>
	{attribute 'OPC.UA.DA' := '1'}  				                
	{attribute 'OPC.UA.DA.Access' := '1'}  				                
	product_condensate_drum_lsh									AT %I*	: BOOL;

    /// <summary>LS-05</summary>
	{attribute 'OPC.UA.DA' := '1'}  				                
	{attribute 'OPC.UA.DA.Access' := '1'}  				                
	condensate_collection_tank_lsl								AT %I*	: BOOL;
    /// <summary>LS-06</summary>
	{attribute 'OPC.UA.DA' := '1'}  				                
	{attribute 'OPC.UA.DA.Access' := '1'}  				                
	condensate_collection_tank_lsh								AT %I*	: BOOL;

	
    /// <summary>B-01</summary>
	{attribute 'OPC.UA.DA' := '1'}  				                
	boiler_package														: BOOL;
    /// <summary>B-01</summary>
	{attribute 'OPC.UA.DA' := '1'}  				                
	{attribute 'OPC.UA.DA.Access' := '1'}  				                
	boiler_package_cmd_status											: BOOL;
    /// <summary>boiler package</summary>
	B_01														AT %Q*	: BOOL;
    /// <summary>B-01</summary>
	{attribute 'OPC.UA.DA' := '1'}  				                
	boiler_ready														: BOOL;

    /// <summary>P_01</summary>
	{attribute 'OPC.UA.DA' := '1'}  				                
	dead_air_vacuum_pump												: BOOL;
    /// <summary>P_01</summary>
	{attribute 'OPC.UA.DA' := '1'}  				                
	{attribute 'OPC.UA.DA.Access' := '1'}  				                
	dead_air_vacuum_pump_cmd_status										: BOOL;
    /// <summary>dead air vacuum pump</summary>
	P_01														AT %Q*	: BOOL;

    /// <summary>P-03</summary>
	{attribute 'OPC.UA.DA' := '1'}  				                
	condensate_collection_tank_pump										: BOOL;
    /// <summary>P-03</summary>
	{attribute 'OPC.UA.DA' := '1'}  				                
	{attribute 'OPC.UA.DA.Access' := '1'}  				                
	condensate_collection_tank_pump_cmd_status							: BOOL;
    /// <summary>condensate collection tank pump</summary>
	P_04														AT %Q*	: BOOL;

    /// <summary>P-04</summary>
	{attribute 'OPC.UA.DA' := '1'}  				                
	product_condensate_pump												: BOOL;
    /// <summary>P-04</summary>
	{attribute 'OPC.UA.DA' := '1'}  				                
	{attribute 'OPC.UA.DA.Access' := '1'}  				                
	product_condensate_pump_cmd_status									: BOOL;
	/// <summary>product condensate pump</summary>
	P_03														AT %Q*	: BOOL;
	

    /// <summary>E-01</summary>
	{attribute 'OPC.UA.DA' := '1'}  				                
	product_condenser													: BOOL;
    /// <summary>E-01</summary>
	{attribute 'OPC.UA.DA' := '1'}  				                
	{attribute 'OPC.UA.DA.Access' := '1'}  				                
	product_condenser_cmd_status										: BOOL;
    /// <summary>product condenser</summary>
	E_01														AT %Q*	: BOOL;

    /// <summary>K_01</summary>
	{attribute 'OPC.UA.DA' := '1'}  				                
	product_blower														: BOOL;
    /// <summary>K_01</summary>
	{attribute 'OPC.UA.DA' := '1'}  				                
	{attribute 'OPC.UA.DA.Access' := '1'}  				                
	product_blower_cmd_status											: BOOL;
    /// <summary>product condenser</summary>
	K_01														AT %Q*	: BOOL;
	
	
	{attribute 'OPC.UA.DA' := '1'}  				                
	product_blower_vfd_enable														: BOOL :=  TRUE;
	{attribute 'OPC.UA.DA' := '1'}  				                
	product_blower_vfd_reset														: BOOL;
	{attribute 'OPC.UA.DA' := '1'}  				                
	{attribute 'OPC.UA.DA.Access' := '1'}  				                
	product_blower_vfd_enabled														: BOOL;
	{attribute 'OPC.UA.DA' := '1'}  				                
	{attribute 'OPC.UA.DA.Access' := '1'}  				                
	product_blower_vfd_error														: BOOL;
	{attribute 'OPC.UA.DA' := '1'}  				                
	product_blower_vfd																: REAL;
	{attribute 'OPC.UA.DA' := '1'}  				                
	{attribute 'OPC.UA.DA.Access' := '1'}  				                
	product_blower_vfd_input														: REAL;
	{attribute 'OPC.UA.DA' := '1'}  				                
	{attribute 'OPC.UA.DA.Access' := '1'}  				                
	product_blower_vfd_output														: REAL;
	product_blower_vfd_control												AT %Q*	: WORD;
	product_blower_vfd_target_vel											AT %Q*	: WORD;
	product_blower_vfd_status												AT %I*	: WORD;
	product_blower_vfd_velocity												AT %I*	: WORD;
	product_blower_vfd_ecat_state											AT %I*  : BOOL;

    /// <summary>C_01</summary>
	{attribute 'OPC.UA.DA' := '1'}  				                
	instrument_air_compressor											: BOOL;
    /// <summary>C_01</summary>
	{attribute 'OPC.UA.DA' := '1'}  				                
	{attribute 'OPC.UA.DA.Access' := '1'}  				                
	instrument_air_compressor_cmd_status								: BOOL;
    /// <summary>product condenser</summary>
	C_01														AT %Q*	: BOOL;

    /// <summary>TB_17</summary>
	{attribute 'OPC.UA.DA' := '1'}  				                
	instrument_air_dryer												: BOOL;
    /// <summary>TB_17</summary>
	{attribute 'OPC.UA.DA' := '1'}  				                
	{attribute 'OPC.UA.DA.Access' := '1'}  				                
	instrument_air_dryer_cmd_status										: BOOL;
    /// <summary>product condenser</summary>
	TB_17														AT %Q*	: BOOL;

    /// <summary>R_01</summary>
	{attribute 'OPC.UA.DA' := '1'}  				                
	radiator															: BOOL;
    /// <summary>R_01</summary>
	{attribute 'OPC.UA.DA' := '1'}  				                
	{attribute 'OPC.UA.DA.Access' := '1'}  				                
	radiator_cmd_status													: BOOL;
    /// <summary>product condenser</summary>
	R_01														AT %Q*	: BOOL;

    /// <summary>AT-01 pump</summary>
	{attribute 'OPC.UA.DA' := '1'}  				                
	dead_air_line_co2_pump												: BOOL;
    /// <summary>AT-01 pump</summary>
	{attribute 'OPC.UA.DA' := '1'}  				                
	{attribute 'OPC.UA.DA.Access' := '1'}  				                
	dead_air_line_co2_pump_cmd_status									: BOOL;
    /// <summary>dead air line co2 pump</summary>
	AT_01_pump													AT %Q*	: BOOL;
	
    /// <summary>AT-01_solenoid</summary>
	{attribute 'OPC.UA.DA' := '1'}  				                
	dead_air_line_co2_sol												: BOOL;
    /// <summary>AT-01_solenoid</summary>
	{attribute 'OPC.UA.DA' := '1'}  				                
	{attribute 'OPC.UA.DA.Access' := '1'}  				                
	dead_air_line_co2_sol_cmd_status									: BOOL;
    /// <summary>dead air CO2 solenoid</summary>
	AT_01_sol													AT %Q*	: BOOL;

	
    /// <summary>AT-01</summary>
	{attribute 'OPC.UA.DA' := '1'}  				                
	{attribute 'OPC.UA.DA.Access' := '1'}  				                
	dead_air_line_co2													: REAL;
    /// <summary>AT-01</summary>
	{attribute 'OPC.UA.DA' := '1'}  				                
	{attribute 'OPC.UA.DA.Access' := '1'}  				                
	dead_air_line_co2_error										AT %I*	: BOOL;
    /// <summary>dead air line co2</summary>
	AT_01														AT %I*	: INT;

    /// <summary>AT-02</summary>
	{attribute 'OPC.UA.DA' := '1'}  				                
	{attribute 'OPC.UA.DA.Access' := '1'}  				                
	product_outlet_co2													: REAL;
    /// <summary>AT-02</summary>
	{attribute 'OPC.UA.DA' := '1'}  				                
	{attribute 'OPC.UA.DA.Access' := '1'}  				                
	product_outlet_co2_error									AT %I*	: BOOL;
    /// <summary>product outlet co2</summary>
	AT_02A														AT %I*	: INT;
    
	/// <summary>AT-07A</summary>
	{attribute 'OPC.UA.DA' := '1'}  				                
	{attribute 'OPC.UA.DA.Access' := '1'}  				                
	product_outlet_h2o													: REAL;
    /// <summary>AT-07A</summary>
	{attribute 'OPC.UA.DA' := '1'}  				                
	{attribute 'OPC.UA.DA.Access' := '1'}  				                
	product_outlet_h2o_error									AT %I*	: BOOL;
	 /// <summary>product outlet h2o</summary>
	AT_07A														AT %I*	: INT;
	
	/// <summary>AT-07B</summary>
	{attribute 'OPC.UA.DA' := '1'}  				                
	{attribute 'OPC.UA.DA.Access' := '1'}  				                
	product_outlet_temperature											: REAL;
    /// <summary>AT-07B</summary>
	{attribute 'OPC.UA.DA' := '1'}  				                
	{attribute 'OPC.UA.DA.Access' := '1'}  				                
	product_outlet_temperature_error							AT %I*	: BOOL;
	 /// <summary>product outlet h2o</summary>
	AT_07B														AT %I*	: INT;
	
  

    /// <summary>AT-03</summary>
	{attribute 'OPC.UA.DA' := '1'}  				                
	{attribute 'OPC.UA.DA.Access' := '1'}  				                
	product_outlet_o2													: REAL;
    /// <summary>AT-03</summary>
	{attribute 'OPC.UA.DA' := '1'}  				                
	{attribute 'OPC.UA.DA.Access' := '1'}  				                
	product_outlet_o2_error										AT %I*	: BOOL;
    /// <summary>product outlet o2</summary>
	AT_03														AT %I*	: INT;
	
	
	/// <summary>AT-02</summary>
	{attribute 'OPC.UA.DA' := '1'}  				                
	{attribute 'OPC.UA.DA.Access' := '1'}  				                
	product_co2sample_h2o												: REAL;
    /// <summary>AT-02</summary>
	{attribute 'OPC.UA.DA' := '1'}  				                
	{attribute 'OPC.UA.DA.Access' := '1'}  				                
	product_co2sample_h2o_error									AT %I*	: BOOL;
	 /// <summary>product outlet h2o</summary>
	AT_02B														AT %I*	: INT;

	
	

    /// <summary>AT-04</summary>
	{attribute 'OPC.UA.DA' := '1'}  				                
	{attribute 'OPC.UA.DA.Access' := '1'}  				                
	condensate_collection_tank_ph										: REAL;
    /// <summary>AT-04</summary>                        
	{attribute 'OPC.UA.DA' := '1'}  				                
	{attribute 'OPC.UA.DA.Access' := '1'}  				            
	condensate_collection_tank_ph_error							AT %I*	: BOOL;
    /// <summary>condensate collection tank ph</summary>
	AT_04														AT %I*	: INT;

    /// <summary>AT-05</summary>
	{attribute 'OPC.UA.DA' := '1'}  				                
	{attribute 'OPC.UA.DA.Access' := '1'}  				                
	condensate_collection_tank_o2										: REAL;
    /// <summary>AT-05</summary>                        
	{attribute 'OPC.UA.DA' := '1'}  				                
	{attribute 'OPC.UA.DA.Access' := '1'}  				            
	condensate_collection_tank_o2_error							AT %I*	: BOOL;
    /// <summary>condensate collection tank o2</summary>
	AT_05														AT %I*	: INT;

    /// <summary>AT-06</summary>
	{attribute 'OPC.UA.DA' := '1'}  				                
	{attribute 'OPC.UA.DA.Access' := '1'}  				                
	condensate_collection_tank_turbidity								: REAL;
    /// <summary>AT-06</summary>                        
	{attribute 'OPC.UA.DA' := '1'}  				                
	{attribute 'OPC.UA.DA.Access' := '1'}  				            
	condensate_collection_tank_turbidity_error					AT %I*	: BOOL;
    /// <summary>condensate collection tank turbidity</summary>
	AT_06														AT %I*	: INT;

    /// <summary>AT-07</summary>
	{attribute 'OPC.UA.DA' := '1'}  				                
	{attribute 'OPC.UA.DA.Access' := '1'}  				                
	weather_humidity													: REAL;
    /// <summary>AT-07</summary>                        
	{attribute 'OPC.UA.DA' := '1'}  				                
	{attribute 'OPC.UA.DA.Access' := '1'}  				            
	weather_humidity_error										AT %I*	: BOOL;
    /// <summary>weather humidity</summary>
	AT_07														AT %I*	: INT;

    /// <summary>FT-01</summary>
	{attribute 'OPC.UA.DA' := '1'}  				                
	{attribute 'OPC.UA.DA.Access' := '1'}  				                
	dead_air_flow														: REAL;
    /// <summary>FT-01</summary>
	{attribute 'OPC.UA.DA' := '1'}  				                
	{attribute 'OPC.UA.DA.Access' := '1'}  				                
	dead_air_flow_error											AT %I*	: BOOL;
    /// <summary>dead air flow</summary>
	FT_01														AT %I*	: INT;

    /// <summary>FT-02</summary>
	{attribute 'OPC.UA.DA' := '1'}  				                
	{attribute 'OPC.UA.DA.Access' := '1'}  				                
	product_outlet_volumetric_flow										: REAL;
	 /// <summary>FT-02</summary>
	{attribute 'OPC.UA.DA' := '1'}  				                
	{attribute 'OPC.UA.DA.Access' := '1'}  				                
	product_outlet_volumetric_flow_total								: REAL;
	/// <summary>FT-02</summary>
	{attribute 'OPC.UA.DA' := '1'}  				                			                
	product_outlet_volumetric_flow_total_enable							: BOOL;
    /// <summary>FT-02</summary>
	{attribute 'OPC.UA.DA' := '1'}  				                
	{attribute 'OPC.UA.DA.Access' := '1'}  				                
	product_outlet_volumetric_flow_error						AT %I*	: BOOL;
    /// <summary>product out volumetric flow</summary>
	FT_03														AT %I*	: INT;

    /// <summary>FT-03</summary>
	{attribute 'OPC.UA.DA' := '1'}  				                
	{attribute 'OPC.UA.DA.Access' := '1'}  					                
	product_outlet_mass_flow											: REAL;
	    /// <summary>FT-03</summary>
	{attribute 'OPC.UA.DA' := '1'}  				                
	{attribute 'OPC.UA.DA.Access' := '1'}  					                
	product_outlet_mass_flow_total										: REAL;
	/// <summary>FT-03</summary>
	{attribute 'OPC.UA.DA' := '1'}  				                					                
	product_outlet_mass_flow_total_enable								: BOOL;
    /// <summary>FT-03</summary>
	{attribute 'OPC.UA.DA' := '1'}  				                
	{attribute 'OPC.UA.DA.Access' := '1'}  				                
	product_outlet_mass_flow_error								AT %I*	: BOOL;
    /// <summary>product outlet mass flow</summary>
	FT_02														AT %I*	: INT;

